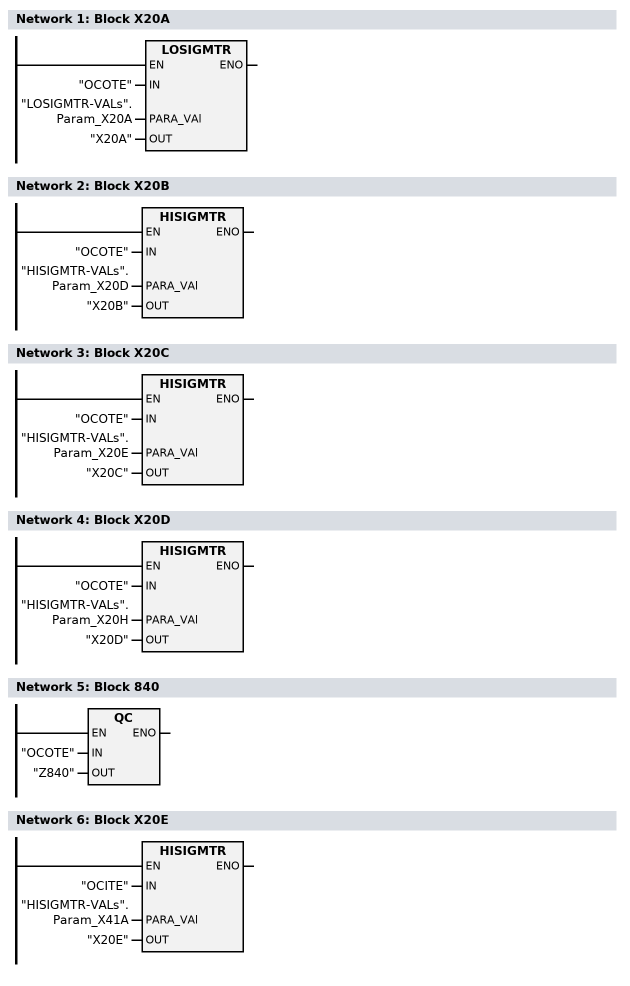
NETWORK
TITLE = Block X20A
      CALL  "LOSIGMTR" (
           IN                       := "OCOTE",
           PARA_VAl                 := "LOSIGMTR-VALs".Param_X20A,
           OUT                      := "X20A");
      NOP   0;
NETWORK
TITLE = Block X20B
      CALL  "HISIGMTR" (
           IN                       := "OCOTE",
           PARA_VAl                 := "HISIGMTR-VALs".Param_X20D,
           OUT                      := "X20B");
      NOP   0;
NETWORK
TITLE = Block X20C
      CALL  "HISIGMTR" (
           IN                       := "OCOTE",
           PARA_VAl                 := "HISIGMTR-VALs".Param_X20E,
           OUT                      := "X20C");
      NOP   0;
NETWORK
TITLE = Block X20D
      CALL  "HISIGMTR" (
           IN                       := "OCOTE",
           PARA_VAl                 := "HISIGMTR-VALs".Param_X20H,
           OUT                      := "X20D");
      NOP   0;
NETWORK
TITLE = Block 840
      CALL  "QC" (
           IN                       := "OCOTE",
           OUT                      := "Z840");
      NOP   0;
NETWORK
TITLE = Block X20E
      CALL  "HISIGMTR" (
           IN                       := "OCITE",
           PARA_VAl                 := "HISIGMTR-VALs".Param_X41A,
           OUT                      := "X20E");
      NOP   0;
END_FUNCTION

FUNCTION "2xHISIGMTV, QC" : VOID	// FC 89
TITLE = 2xHISIGMTV, QC
//Supporting block for sheet 12 (ATC)
AUTHOR : RJ
VERSION : 0.0
VAR_INPUT
  INPUT : REAL ;
  STPT_1 : REAL ;
  STPT_2 : REAL ;
  Param_1 : STRUCT
   DBAN : REAL ;
  END_STRUCT ;
  Param_2 : STRUCT
   DBAN : REAL ;
  END_STRUCT ;
END_VAR
VAR_OUTPUT
  OUT_1 : BOOL ;
  OUT_2 : BOOL ;
  OUT_QC : BOOL ;
END_VAR
VAR_TEMP
  Para_1 : STRUCT
   DBAN : REAL ;
  END_STRUCT ;
  Para_2 : STRUCT
   DBAN : REAL ;
  END_STRUCT ;
END_VAR
BEGIN
// body was compiled from an SCL source; compiled code not shown
END_FUNCTION

FUNCTION "Sheet 12 (ATC)" : VOID	// FC 91
TITLE = Sheet 12 (ATC)
//BEARING METAL TEMPERATURES (Analog)
AUTHOR : RJ
FAMILY : ATC
VERSION : 0.1
BEGIN
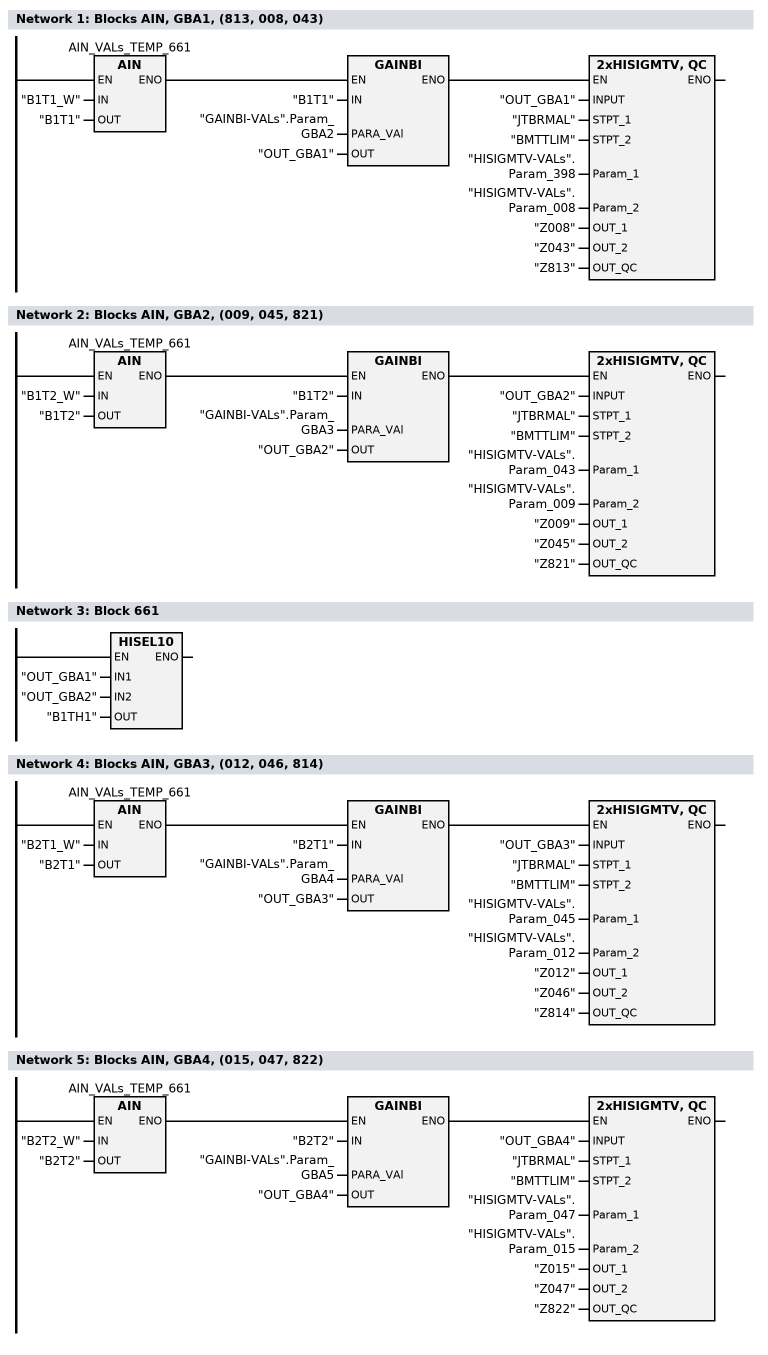
NETWORK
TITLE = Blocks AIN, GBA1, (813, 008, 043)
      A(;
      A(;
      CALL  "AIN" , "AIN_VALs_TEMP_661" (
           IN                       := "B1T1_W",
           OUT                      := "B1T1");
      A     BR;
      );
      JNB   _001;
      CALL  "GAINBI" (
           IN                       := "B1T1",
           PARA_VAl                 := "GAINBI-VALs".Param_GBA2,
           OUT                      := "OUT_GBA1");
_001: A     BR;
      );
      JNB   _002;
      CALL  "2xHISIGMTV, QC" (
           INPUT                    := "OUT_GBA1",
           STPT_1                   := "JTBRMAL",
           STPT_2                   := "BMTTLIM",
           Param_1                  := "HISIGMTV-VALs".Param_398,
           Param_2                  := "HISIGMTV-VALs".Param_008,
           OUT_1                    := "Z008",
           OUT_2                    := "Z043",
           OUT_QC                   := "Z813");
_002: NOP   0;
NETWORK
TITLE = Blocks AIN, GBA2, (009, 045, 821)
      A(;
      A(;
      CALL  "AIN" , "AIN_VALs_TEMP_661" (
           IN                       := "B1T2_W",
           OUT                      := "B1T2");
      A     BR;
      );
      JNB   _003;
      CALL  "GAINBI" (
           IN                       := "B1T2",
           PARA_VAl                 := "GAINBI-VALs".Param_GBA3,
           OUT                      := "OUT_GBA2");
_003: A     BR;
      );
      JNB   _004;
      CALL  "2xHISIGMTV, QC" (
           INPUT                    := "OUT_GBA2",
           STPT_1                   := "JTBRMAL",
           STPT_2                   := "BMTTLIM",
           Param_1                  := "HISIGMTV-VALs".Param_043,
           Param_2                  := "HISIGMTV-VALs".Param_009,
           OUT_1                    := "Z009",
           OUT_2                    := "Z045",
           OUT_QC                   := "Z821");
_004: NOP   0;
NETWORK
TITLE = Block 661
      CALL  "HISEL10" (
           IN1                      := "OUT_GBA1",
           IN2                      := "OUT_GBA2",
           OUT                      := "B1TH1");
      NOP   0;
NETWORK
TITLE = Blocks AIN, GBA3, (012, 046, 814)
      A(;
      A(;
      CALL  "AIN" , "AIN_VALs_TEMP_661" (
           IN                       := "B2T1_W",
           OUT                      := "B2T1");
      A     BR;
      );
      JNB   _005;
      CALL  "GAINBI" (
           IN                       := "B2T1",
           PARA_VAl                 := "GAINBI-VALs".Param_GBA4,
           OUT                      := "OUT_GBA3");
_005: A     BR;
      );
      JNB   _006;
      CALL  "2xHISIGMTV, QC" (
           INPUT                    := "OUT_GBA3",
           STPT_1                   := "JTBRMAL",
           STPT_2                   := "BMTTLIM",
           Param_1                  := "HISIGMTV-VALs".Param_045,
           Param_2                  := "HISIGMTV-VALs".Param_012,
           OUT_1                    := "Z012",
           OUT_2                    := "Z046",
           OUT_QC                   := "Z814");
_006: NOP   0;
NETWORK
TITLE = Blocks AIN, GBA4, (015, 047, 822)
      A(;
      A(;
      CALL  "AIN" , "AIN_VALs_TEMP_661" (
           IN                       := "B2T2_W",
           OUT                      := "B2T2");
      A     BR;
      );
      JNB   _007;
      CALL  "GAINBI" (
           IN                       := "B2T2",
           PARA_VAl                 := "GAINBI-VALs".Param_GBA5,
           OUT                      := "OUT_GBA4");
_007: A     BR;
      );
      JNB   _008;
      CALL  "2xHISIGMTV, QC" (
           INPUT                    := "OUT_GBA4",
           STPT_1                   := "JTBRMAL",
           STPT_2                   := "BMTTLIM",
           Param_1                  := "HISIGMTV-VALs".Param_047,
           Param_2                  := "HISIGMTV-VALs".Param_015,
           OUT_1                    := "Z015",
           OUT_2                    := "Z047",
           OUT_QC                   := "Z822");
_008: NOP   0;
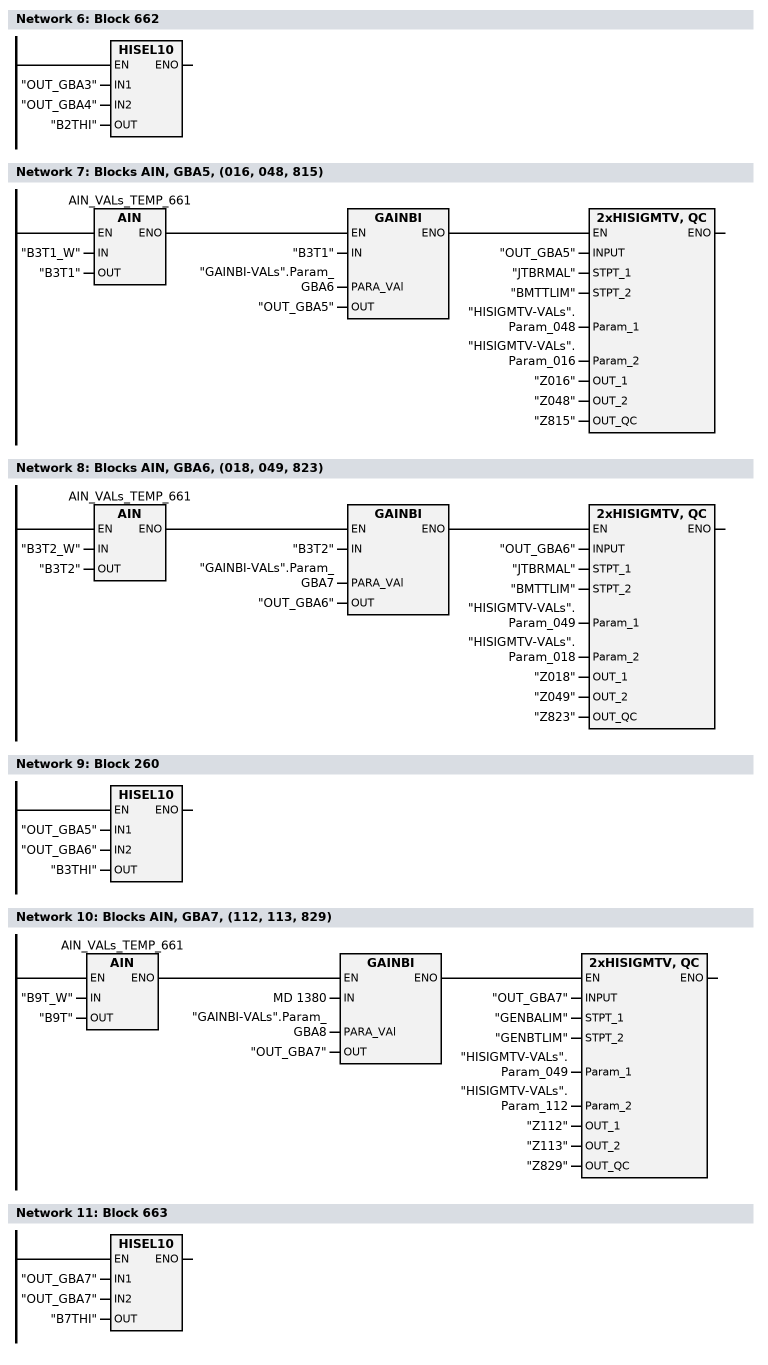
NETWORK
TITLE = Block 662
      CALL  "HISEL10" (
           IN1                      := "OUT_GBA3",
           IN2                      := "OUT_GBA4",
           OUT                      := "B2THI");
      NOP   0;
NETWORK
TITLE = Blocks AIN, GBA5, (016, 048, 815)
      A(;
      A(;
      CALL  "AIN" , "AIN_VALs_TEMP_661" (
           IN                       := "B3T1_W",
           OUT                      := "B3T1");
      A     BR;
      );
      JNB   _009;
      CALL  "GAINBI" (
           IN                       := "B3T1",
           PARA_VAl                 := "GAINBI-VALs".Param_GBA6,
           OUT                      := "OUT_GBA5");
_009: A     BR;
      );
      JNB   _00a;
      CALL  "2xHISIGMTV, QC" (
           INPUT                    := "OUT_GBA5",
           STPT_1                   := "JTBRMAL",
           STPT_2                   := "BMTTLIM",
           Param_1                  := "HISIGMTV-VALs".Param_048,
           Param_2                  := "HISIGMTV-VALs".Param_016,
           OUT_1                    := "Z016",
           OUT_2                    := "Z048",
           OUT_QC                   := "Z815");
_00a: NOP   0;
NETWORK
TITLE = Blocks AIN, GBA6, (018, 049, 823)
      A(;
      A(;
      CALL  "AIN" , "AIN_VALs_TEMP_661" (
           IN                       := "B3T2_W",
           OUT                      := "B3T2");
      A     BR;
      );
      JNB   _00b;
      CALL  "GAINBI" (
           IN                       := "B3T2",
           PARA_VAl                 := "GAINBI-VALs".Param_GBA7,
           OUT                      := "OUT_GBA6");
_00b: A     BR;
      );
      JNB   _00c;
      CALL  "2xHISIGMTV, QC" (
           INPUT                    := "OUT_GBA6",
           STPT_1                   := "JTBRMAL",
           STPT_2                   := "BMTTLIM",
           Param_1                  := "HISIGMTV-VALs".Param_049,
           Param_2                  := "HISIGMTV-VALs".Param_018,
           OUT_1                    := "Z018",
           OUT_2                    := "Z049",
           OUT_QC                   := "Z823");
_00c: NOP   0;
NETWORK
TITLE = Block 260
      CALL  "HISEL10" (
           IN1                      := "OUT_GBA5",
           IN2                      := "OUT_GBA6",
           OUT                      := "B3THI");
      NOP   0;
NETWORK
TITLE = Blocks AIN, GBA7, (112, 113, 829)
      A(;
      A(;
      CALL  "AIN" , "AIN_VALs_TEMP_661" (
           IN                       := "B9T_W",
           OUT                      := "B9T");
      A     BR;
      );
      JNB   _00d;
      CALL  "GAINBI" (
           IN                       := MD 1380,
           PARA_VAl                 := "GAINBI-VALs".Param_GBA8,
           OUT                      := "OUT_GBA7");
_00d: A     BR;
      );
      JNB   _00e;
      CALL  "2xHISIGMTV, QC" (
           INPUT                    := "OUT_GBA7",
           STPT_1                   := "GENBALIM",
           STPT_2                   := "GENBTLIM",
           Param_1                  := "HISIGMTV-VALs".Param_049,
           Param_2                  := "HISIGMTV-VALs".Param_112,
           OUT_1                    := "Z112",
           OUT_2                    := "Z113",
           OUT_QC                   := "Z829");
_00e: NOP   0;
NETWORK
TITLE = Block 663
      CALL  "HISEL10" (
           IN1                      := "OUT_GBA7",
           IN2                      := "OUT_GBA7",
           OUT                      := "B7THI");
      NOP   0;
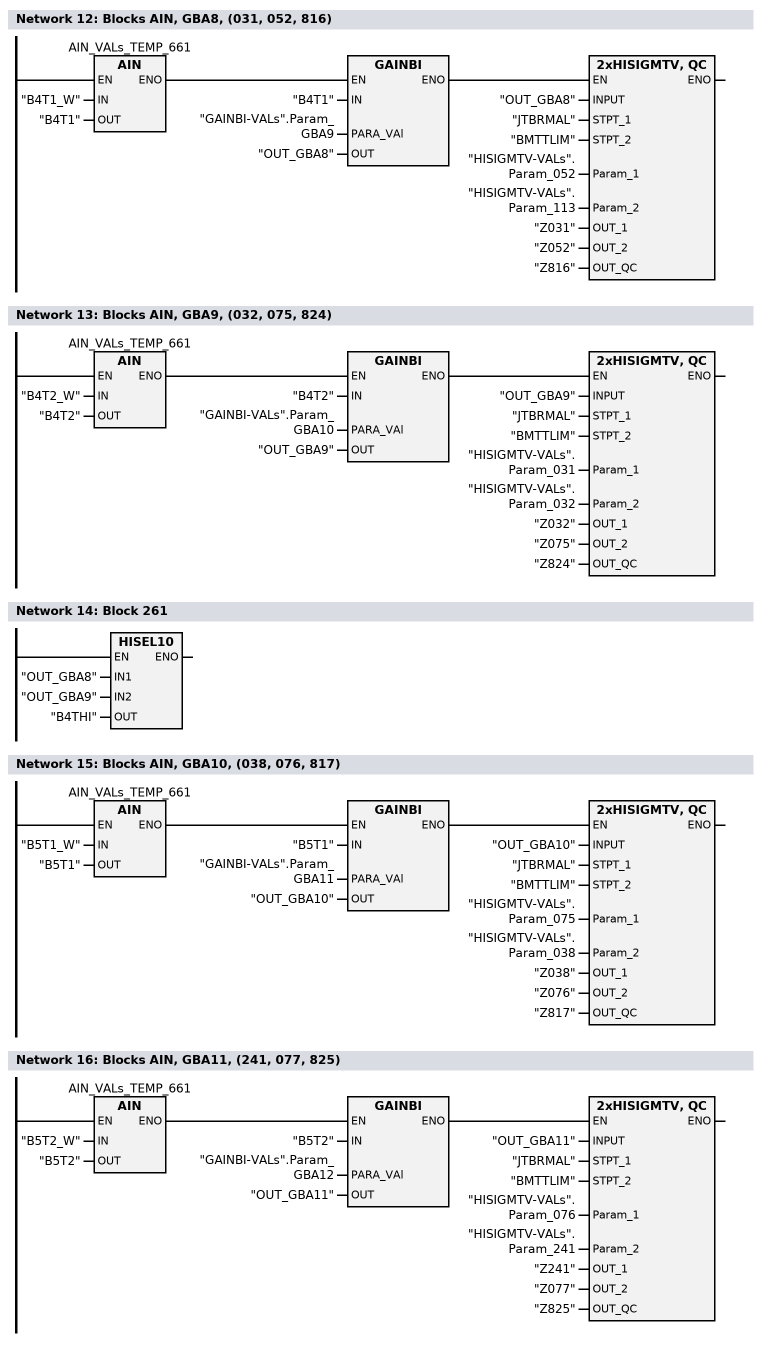
NETWORK
TITLE = Blocks AIN, GBA8, (031, 052, 816)
      A(;
      A(;
      CALL  "AIN" , "AIN_VALs_TEMP_661" (
           IN                       := "B4T1_W",
           OUT                      := "B4T1");
      A     BR;
      );
      JNB   _00f;
      CALL  "GAINBI" (
           IN                       := "B4T1",
           PARA_VAl                 := "GAINBI-VALs".Param_GBA9,
           OUT                      := "OUT_GBA8");
_00f: A     BR;
      );
      JNB   _010;
      CALL  "2xHISIGMTV, QC" (
           INPUT                    := "OUT_GBA8",
           STPT_1                   := "JTBRMAL",
           STPT_2                   := "BMTTLIM",
           Param_1                  := "HISIGMTV-VALs".Param_052,
           Param_2                  := "HISIGMTV-VALs".Param_113,
           OUT_1                    := "Z031",
           OUT_2                    := "Z052",
           OUT_QC                   := "Z816");
_010: NOP   0;
NETWORK
TITLE = Blocks AIN, GBA9, (032, 075, 824)
      A(;
      A(;
      CALL  "AIN" , "AIN_VALs_TEMP_661" (
           IN                       := "B4T2_W",
           OUT                      := "B4T2");
      A     BR;
      );
      JNB   _011;
      CALL  "GAINBI" (
           IN                       := "B4T2",
           PARA_VAl                 := "GAINBI-VALs".Param_GBA10,
           OUT                      := "OUT_GBA9");
_011: A     BR;
      );
      JNB   _012;
      CALL  "2xHISIGMTV, QC" (
           INPUT                    := "OUT_GBA9",
           STPT_1                   := "JTBRMAL",
           STPT_2                   := "BMTTLIM",
           Param_1                  := "HISIGMTV-VALs".Param_031,
           Param_2                  := "HISIGMTV-VALs".Param_032,
           OUT_1                    := "Z032",
           OUT_2                    := "Z075",
           OUT_QC                   := "Z824");
_012: NOP   0;
NETWORK
TITLE = Block 261
      CALL  "HISEL10" (
           IN1                      := "OUT_GBA8",
           IN2                      := "OUT_GBA9",
           OUT                      := "B4THI");
      NOP   0;
NETWORK
TITLE = Blocks AIN, GBA10, (038, 076, 817)
      A(;
      A(;
      CALL  "AIN" , "AIN_VALs_TEMP_661" (
           IN                       := "B5T1_W",
           OUT                      := "B5T1");
      A     BR;
      );
      JNB   _013;
      CALL  "GAINBI" (
           IN                       := "B5T1",
           PARA_VAl                 := "GAINBI-VALs".Param_GBA11,
           OUT                      := "OUT_GBA10");
_013: A     BR;
      );
      JNB   _014;
      CALL  "2xHISIGMTV, QC" (
           INPUT                    := "OUT_GBA10",
           STPT_1                   := "JTBRMAL",
           STPT_2                   := "BMTTLIM",
           Param_1                  := "HISIGMTV-VALs".Param_075,
           Param_2                  := "HISIGMTV-VALs".Param_038,
           OUT_1                    := "Z038",
           OUT_2                    := "Z076",
           OUT_QC                   := "Z817");
_014: NOP   0;
NETWORK
TITLE = Blocks AIN, GBA11, (241, 077, 825)
      A(;
      A(;
      CALL  "AIN" , "AIN_VALs_TEMP_661" (
           IN                       := "B5T2_W",
           OUT                      := "B5T2");
      A     BR;
      );
      JNB   _015;
      CALL  "GAINBI" (
           IN                       := "B5T2",
           PARA_VAl                 := "GAINBI-VALs".Param_GBA12,
           OUT                      := "OUT_GBA11");
_015: A     BR;
      );
      JNB   _016;
      CALL  "2xHISIGMTV, QC" (
           INPUT                    := "OUT_GBA11",
           STPT_1                   := "JTBRMAL",
           STPT_2                   := "BMTTLIM",
           Param_1                  := "HISIGMTV-VALs".Param_076,
           Param_2                  := "HISIGMTV-VALs".Param_241,
           OUT_1                    := "Z241",
           OUT_2                    := "Z077",
           OUT_QC                   := "Z825");
_016: NOP   0;
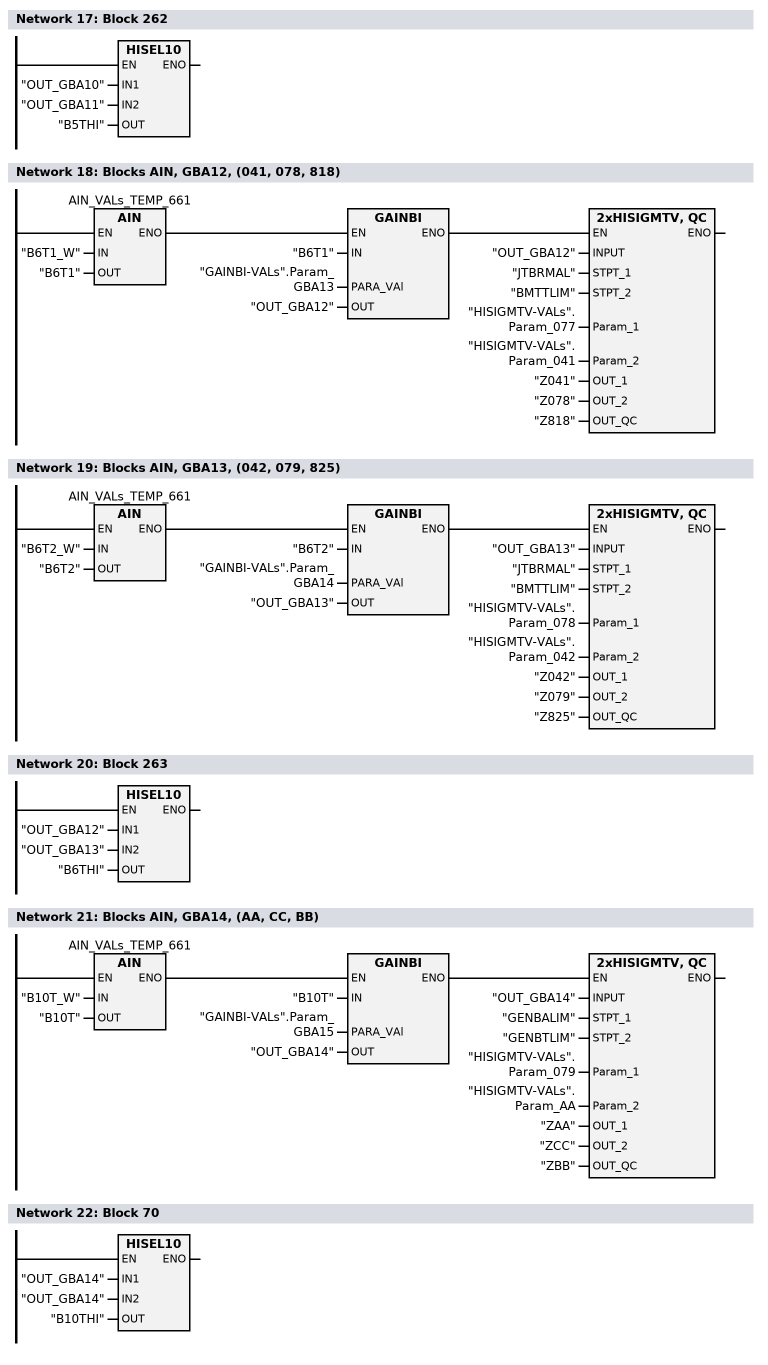
NETWORK
TITLE = Block 262
      CALL  "HISEL10" (
           IN1                      := "OUT_GBA10",
           IN2                      := "OUT_GBA11",
           OUT                      := "B5THI");
      NOP   0;
NETWORK
TITLE = Blocks AIN, GBA12, (041, 078, 818)
      A(;
      A(;
      CALL  "AIN" , "AIN_VALs_TEMP_661" (
           IN                       := "B6T1_W",
           OUT                      := "B6T1");
      A     BR;
      );
      JNB   _017;
      CALL  "GAINBI" (
           IN                       := "B6T1",
           PARA_VAl                 := "GAINBI-VALs".Param_GBA13,
           OUT                      := "OUT_GBA12");
_017: A     BR;
      );
      JNB   _018;
      CALL  "2xHISIGMTV, QC" (
           INPUT                    := "OUT_GBA12",
           STPT_1                   := "JTBRMAL",
           STPT_2                   := "BMTTLIM",
           Param_1                  := "HISIGMTV-VALs".Param_077,
           Param_2                  := "HISIGMTV-VALs".Param_041,
           OUT_1                    := "Z041",
           OUT_2                    := "Z078",
           OUT_QC                   := "Z818");
_018: NOP   0;
NETWORK
TITLE = Blocks AIN, GBA13, (042, 079, 825)
      A(;
      A(;
      CALL  "AIN" , "AIN_VALs_TEMP_661" (
           IN                       := "B6T2_W",
           OUT                      := "B6T2");
      A     BR;
      );
      JNB   _019;
      CALL  "GAINBI" (
           IN                       := "B6T2",
           PARA_VAl                 := "GAINBI-VALs".Param_GBA14,
           OUT                      := "OUT_GBA13");
_019: A     BR;
      );
      JNB   _01a;
      CALL  "2xHISIGMTV, QC" (
           INPUT                    := "OUT_GBA13",
           STPT_1                   := "JTBRMAL",
           STPT_2                   := "BMTTLIM",
           Param_1                  := "HISIGMTV-VALs".Param_078,
           Param_2                  := "HISIGMTV-VALs".Param_042,
           OUT_1                    := "Z042",
           OUT_2                    := "Z079",
           OUT_QC                   := "Z825");
_01a: NOP   0;
NETWORK
TITLE = Block 263
      CALL  "HISEL10" (
           IN1                      := "OUT_GBA12",
           IN2                      := "OUT_GBA13",
           OUT                      := "B6THI");
      NOP   0;
NETWORK
TITLE = Blocks AIN, GBA14, (AA, CC, BB)
      A(;
      A(;
      CALL  "AIN" , "AIN_VALs_TEMP_661" (
           IN                       := "B10T_W",
           OUT                      := "B10T");
      A     BR;
      );
      JNB   _01b;
      CALL  "GAINBI" (
           IN                       := "B10T",
           PARA_VAl                 := "GAINBI-VALs".Param_GBA15,
           OUT                      := "OUT_GBA14");
_01b: A     BR;
      );
      JNB   _01c;
      CALL  "2xHISIGMTV, QC" (
           INPUT                    := "OUT_GBA14",
           STPT_1                   := "GENBALIM",
           STPT_2                   := "GENBTLIM",
           Param_1                  := "HISIGMTV-VALs".Param_079,
           Param_2                  := "HISIGMTV-VALs".Param_AA,
           OUT_1                    := "ZAA",
           OUT_2                    := "ZCC",
           OUT_QC                   := "ZBB");
_01c: NOP   0;
NETWORK
TITLE = Block 70
      CALL  "HISEL10" (
           IN1                      := "OUT_GBA14",
           IN2                      := "OUT_GBA14",
           OUT                      := "B10THI");
      NOP   0;
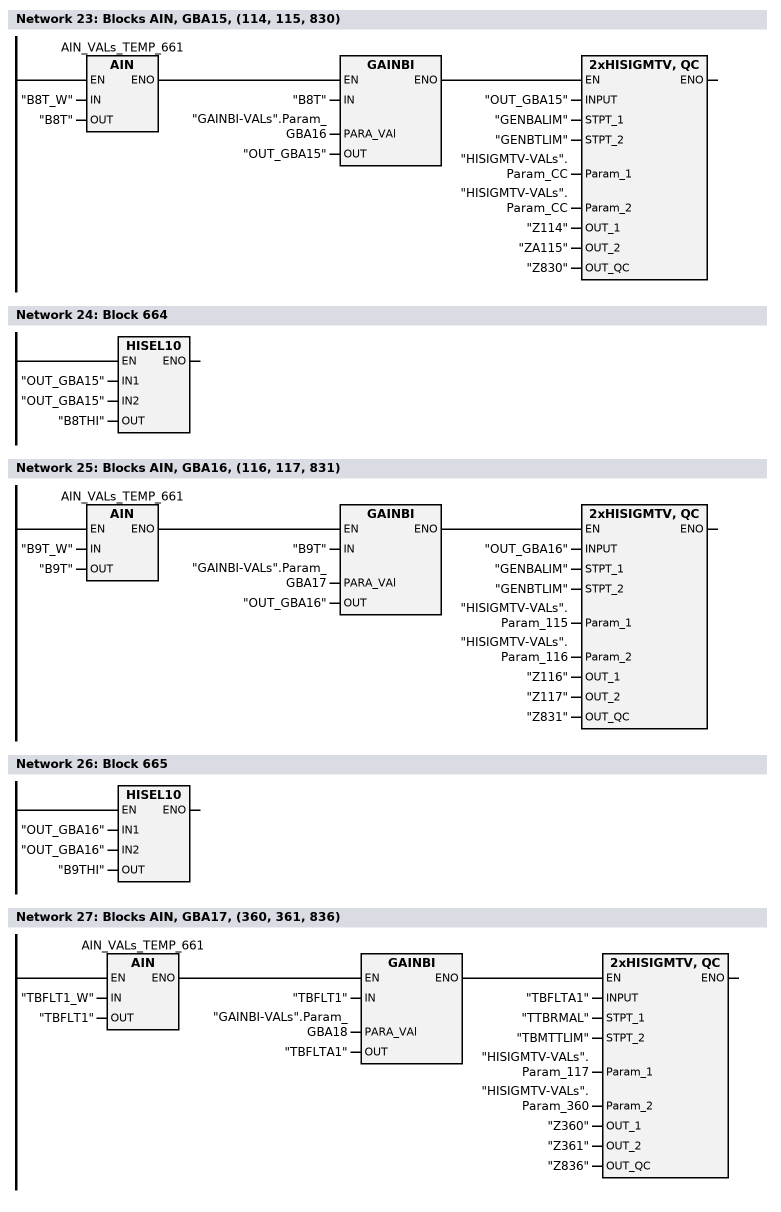
NETWORK
TITLE = Blocks AIN, GBA15, (114, 115, 830)
      A(;
      A(;
      CALL  "AIN" , "AIN_VALs_TEMP_661" (
           IN                       := "B8T_W",
           OUT                      := "B8T");
      A     BR;
      );
      JNB   _01d;
      CALL  "GAINBI" (
           IN                       := "B8T",
           PARA_VAl                 := "GAINBI-VALs".Param_GBA16,
           OUT                      := "OUT_GBA15");
_01d: A     BR;
      );
      JNB   _01e;
      CALL  "2xHISIGMTV, QC" (
           INPUT                    := "OUT_GBA15",
           STPT_1                   := "GENBALIM",
           STPT_2                   := "GENBTLIM",
           Param_1                  := "HISIGMTV-VALs".Param_CC,
           Param_2                  := "HISIGMTV-VALs".Param_CC,
           OUT_1                    := "Z114",
           OUT_2                    := "ZA115",
           OUT_QC                   := "Z830");
_01e: NOP   0;
NETWORK
TITLE = Block 664
      CALL  "HISEL10" (
           IN1                      := "OUT_GBA15",
           IN2                      := "OUT_GBA15",
           OUT                      := "B8THI");
      NOP   0;
NETWORK
TITLE = Blocks AIN, GBA16, (116, 117, 831)
      A(;
      A(;
      CALL  "AIN" , "AIN_VALs_TEMP_661" (
           IN                       := "B9T_W",
           OUT                      := "B9T");
      A     BR;
      );
      JNB   _01f;
      CALL  "GAINBI" (
           IN                       := "B9T",
           PARA_VAl                 := "GAINBI-VALs".Param_GBA17,
           OUT                      := "OUT_GBA16");
_01f: A     BR;
      );
      JNB   _020;
      CALL  "2xHISIGMTV, QC" (
           INPUT                    := "OUT_GBA16",
           STPT_1                   := "GENBALIM",
           STPT_2                   := "GENBTLIM",
           Param_1                  := "HISIGMTV-VALs".Param_115,
           Param_2                  := "HISIGMTV-VALs".Param_116,
           OUT_1                    := "Z116",
           OUT_2                    := "Z117",
           OUT_QC                   := "Z831");
_020: NOP   0;
NETWORK
TITLE = Block 665
      CALL  "HISEL10" (
           IN1                      := "OUT_GBA16",
           IN2                      := "OUT_GBA16",
           OUT                      := "B9THI");
      NOP   0;
NETWORK
TITLE = Blocks AIN, GBA17, (360, 361, 836)
      A(;
      A(;
      CALL  "AIN" , "AIN_VALs_TEMP_661" (
           IN                       := "TBFLT1_W",
           OUT                      := "TBFLT1");
      A     BR;
      );
      JNB   _021;
      CALL  "GAINBI" (
           IN                       := "TBFLT1",
           PARA_VAl                 := "GAINBI-VALs".Param_GBA18,
           OUT                      := "TBFLTA1");
_021: A     BR;
      );
      JNB   _022;
      CALL  "2xHISIGMTV, QC" (
           INPUT                    := "TBFLTA1",
           STPT_1                   := "TTBRMAL",
           STPT_2                   := "TBMTTLIM",
           Param_1                  := "HISIGMTV-VALs".Param_117,
           Param_2                  := "HISIGMTV-VALs".Param_360,
           OUT_1                    := "Z360",
           OUT_2                    := "Z361",
           OUT_QC                   := "Z836");
_022: NOP   0;
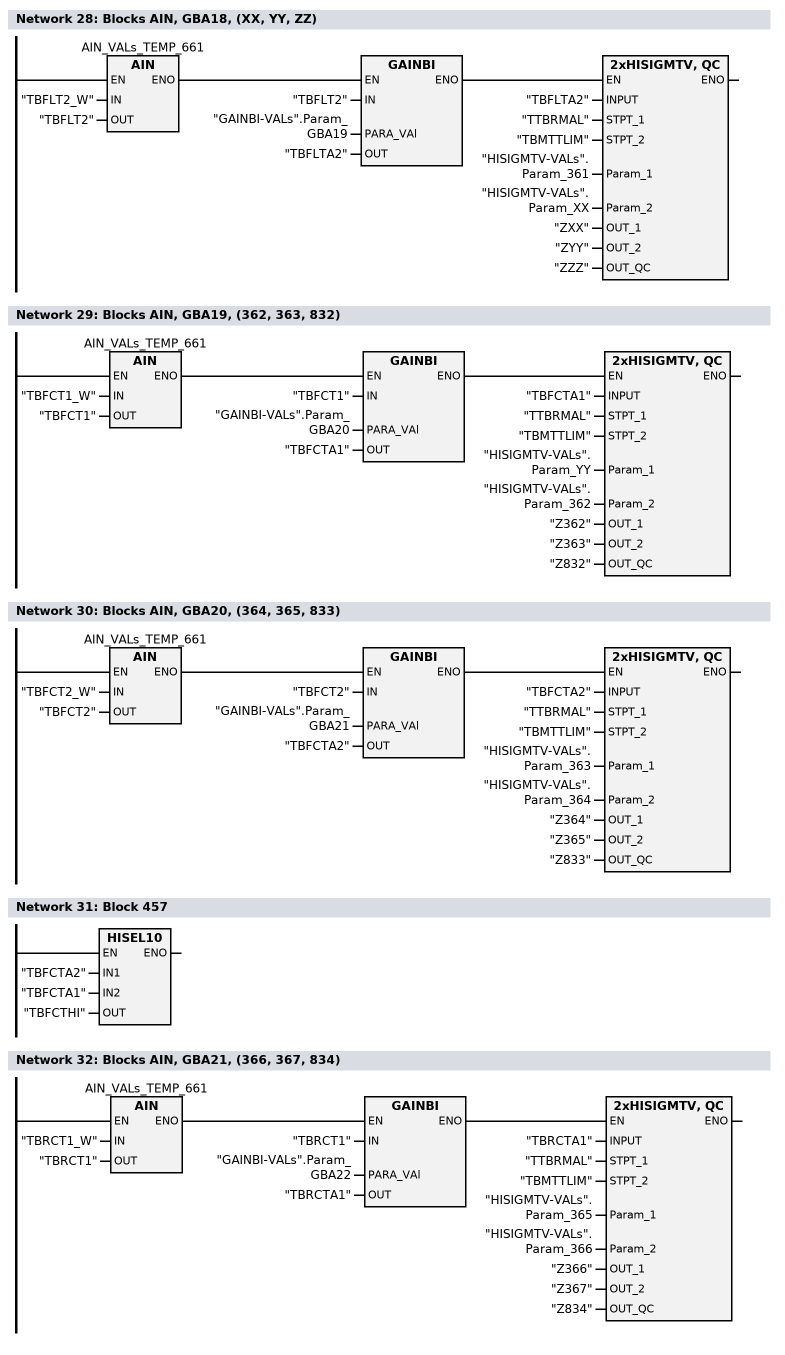
NETWORK
TITLE = Blocks AIN, GBA18, (XX, YY, ZZ)
      A(;
      A(;
      CALL  "AIN" , "AIN_VALs_TEMP_661" (
           IN                       := "TBFLT2_W",
           OUT                      := "TBFLT2");
      A     BR;
      );
      JNB   _023;
      CALL  "GAINBI" (
           IN                       := "TBFLT2",
           PARA_VAl                 := "GAINBI-VALs".Param_GBA19,
           OUT                      := "TBFLTA2");
_023: A     BR;
      );
      JNB   _024;
      CALL  "2xHISIGMTV, QC" (
           INPUT                    := "TBFLTA2",
           STPT_1                   := "TTBRMAL",
           STPT_2                   := "TBMTTLIM",
           Param_1                  := "HISIGMTV-VALs".Param_361,
           Param_2                  := "HISIGMTV-VALs".Param_XX,
           OUT_1                    := "ZXX",
           OUT_2                    := "ZYY",
           OUT_QC                   := "ZZZ");
_024: NOP   0;
NETWORK
TITLE = Blocks AIN, GBA19, (362, 363, 832)
      A(;
      A(;
      CALL  "AIN" , "AIN_VALs_TEMP_661" (
           IN                       := "TBFCT1_W",
           OUT                      := "TBFCT1");
      A     BR;
      );
      JNB   _025;
      CALL  "GAINBI" (
           IN                       := "TBFCT1",
           PARA_VAl                 := "GAINBI-VALs".Param_GBA20,
           OUT                      := "TBFCTA1");
_025: A     BR;
      );
      JNB   _026;
      CALL  "2xHISIGMTV, QC" (
           INPUT                    := "TBFCTA1",
           STPT_1                   := "TTBRMAL",
           STPT_2                   := "TBMTTLIM",
           Param_1                  := "HISIGMTV-VALs".Param_YY,
           Param_2                  := "HISIGMTV-VALs".Param_362,
           OUT_1                    := "Z362",
           OUT_2                    := "Z363",
           OUT_QC                   := "Z832");
_026: NOP   0;
NETWORK
TITLE = Blocks AIN, GBA20, (364, 365, 833)
      A(;
      A(;
      CALL  "AIN" , "AIN_VALs_TEMP_661" (
           IN                       := "TBFCT2_W",
           OUT                      := "TBFCT2");
      A     BR;
      );
      JNB   _027;
      CALL  "GAINBI" (
           IN                       := "TBFCT2",
           PARA_VAl                 := "GAINBI-VALs".Param_GBA21,
           OUT                      := "TBFCTA2");
_027: A     BR;
      );
      JNB   _028;
      CALL  "2xHISIGMTV, QC" (
           INPUT                    := "TBFCTA2",
           STPT_1                   := "TTBRMAL",
           STPT_2                   := "TBMTTLIM",
           Param_1                  := "HISIGMTV-VALs".Param_363,
           Param_2                  := "HISIGMTV-VALs".Param_364,
           OUT_1                    := "Z364",
           OUT_2                    := "Z365",
           OUT_QC                   := "Z833");
_028: NOP   0;
NETWORK
TITLE = Block 457
      CALL  "HISEL10" (
           IN1                      := "TBFCTA2",
           IN2                      := "TBFCTA1",
           OUT                      := "TBFCTHI");
      NOP   0;
NETWORK
TITLE = Blocks AIN, GBA21, (366, 367, 834)
      A(;
      A(;
      CALL  "AIN" , "AIN_VALs_TEMP_661" (
           IN                       := "TBRCT1_W",
           OUT                      := "TBRCT1");
      A     BR;
      );
      JNB   _029;
      CALL  "GAINBI" (
           IN                       := "TBRCT1",
           PARA_VAl                 := "GAINBI-VALs".Param_GBA22,
           OUT                      := "TBRCTA1");
_029: A     BR;
      );
      JNB   _02a;
      CALL  "2xHISIGMTV, QC" (
           INPUT                    := "TBRCTA1",
           STPT_1                   := "TTBRMAL",
           STPT_2                   := "TBMTTLIM",
           Param_1                  := "HISIGMTV-VALs".Param_365,
           Param_2                  := "HISIGMTV-VALs".Param_366,
           OUT_1                    := "Z366",
           OUT_2                    := "Z367",
           OUT_QC                   := "Z834");
_02a: NOP   0;
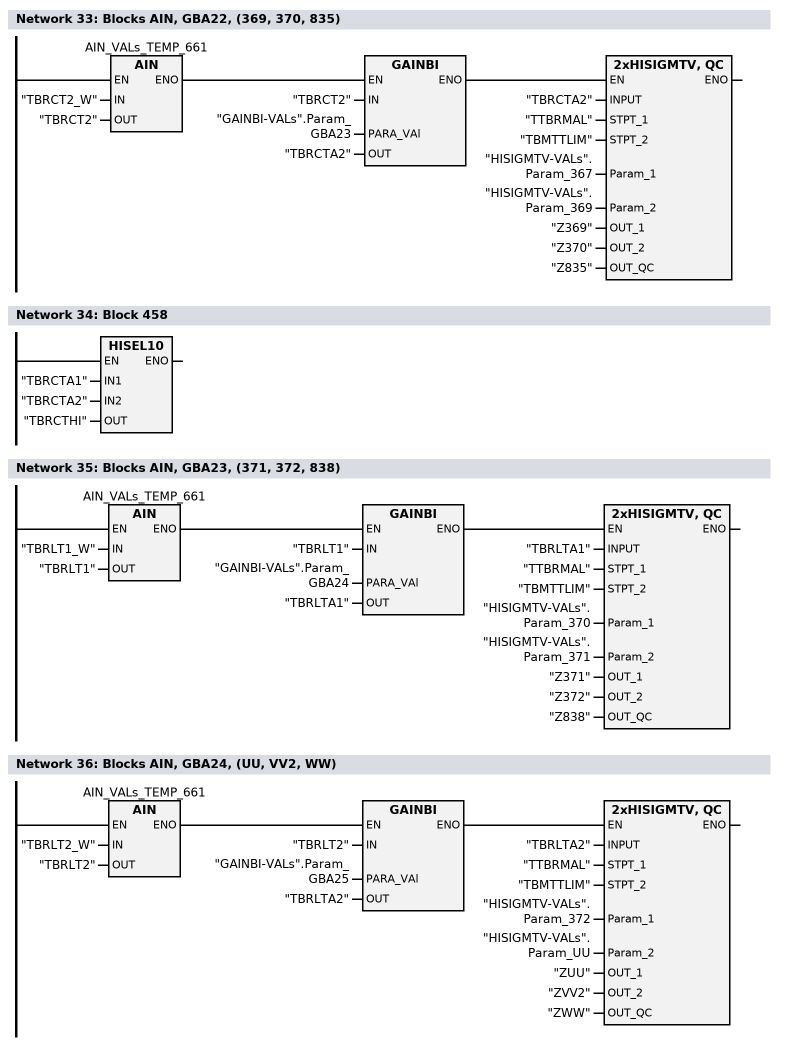
NETWORK
TITLE = Blocks AIN, GBA22, (369, 370, 835)
      A(;
      A(;
      CALL  "AIN" , "AIN_VALs_TEMP_661" (
           IN                       := "TBRCT2_W",
           OUT                      := "TBRCT2");
      A     BR;
      );
      JNB   _02b;
      CALL  "GAINBI" (
           IN                       := "TBRCT2",
           PARA_VAl                 := "GAINBI-VALs".Param_GBA23,
           OUT                      := "TBRCTA2");
_02b: A     BR;
      );
      JNB   _02c;
      CALL  "2xHISIGMTV, QC" (
           INPUT                    := "TBRCTA2",
           STPT_1                   := "TTBRMAL",
           STPT_2                   := "TBMTTLIM",
           Param_1                  := "HISIGMTV-VALs".Param_367,
           Param_2                  := "HISIGMTV-VALs".Param_369,
           OUT_1                    := "Z369",
           OUT_2                    := "Z370",
           OUT_QC                   := "Z835");
_02c: NOP   0;
NETWORK
TITLE = Block 458
      CALL  "HISEL10" (
           IN1                      := "TBRCTA1",
           IN2                      := "TBRCTA2",
           OUT                      := "TBRCTHI");
      NOP   0;
NETWORK
TITLE = Blocks AIN, GBA23, (371, 372, 838)
      A(;
      A(;
      CALL  "AIN" , "AIN_VALs_TEMP_661" (
           IN                       := "TBRLT1_W",
           OUT                      := "TBRLT1");
      A     BR;
      );
      JNB   _02d;
      CALL  "GAINBI" (
           IN                       := "TBRLT1",
           PARA_VAl                 := "GAINBI-VALs".Param_GBA24,
           OUT                      := "TBRLTA1");
_02d: A     BR;
      );
      JNB   _02e;
      CALL  "2xHISIGMTV, QC" (
           INPUT                    := "TBRLTA1",
           STPT_1                   := "TTBRMAL",
           STPT_2                   := "TBMTTLIM",
           Param_1                  := "HISIGMTV-VALs".Param_370,
           Param_2                  := "HISIGMTV-VALs".Param_371,
           OUT_1                    := "Z371",
           OUT_2                    := "Z372",
           OUT_QC                   := "Z838");
_02e: NOP   0;
NETWORK
TITLE = Blocks AIN, GBA24, (UU, VV2, WW)
      A(;
      A(;
      CALL  "AIN" , "AIN_VALs_TEMP_661" (
           IN                       := "TBRLT2_W",
           OUT                      := "TBRLT2");
      A     BR;
      );
      JNB   _02f;
      CALL  "GAINBI" (
           IN                       := "TBRLT2",
           PARA_VAl                 := "GAINBI-VALs".Param_GBA25,
           OUT                      := "TBRLTA2");
_02f: A     BR;
      );
      JNB   _030;
      CALL  "2xHISIGMTV, QC" (
           INPUT                    := "TBRLTA2",
           STPT_1                   := "TTBRMAL",
           STPT_2                   := "TBMTTLIM",
           Param_1                  := "HISIGMTV-VALs".Param_372,
           Param_2                  := "HISIGMTV-VALs".Param_UU,
           OUT_1                    := "ZUU",
           OUT_2                    := "ZVV2",
           OUT_QC                   := "ZWW");
_030: NOP   0;
END_FUNCTION

FUNCTION "Sheet 13 (ATC)" : VOID	// FC 92
TITLE = Sheet 13 (ATC)
//BEARING METAL, OIL COOLER - P08MXX (Digital)
AUTHOR : RJ
FAMILY : ATC
VERSION : 0.1
BEGIN
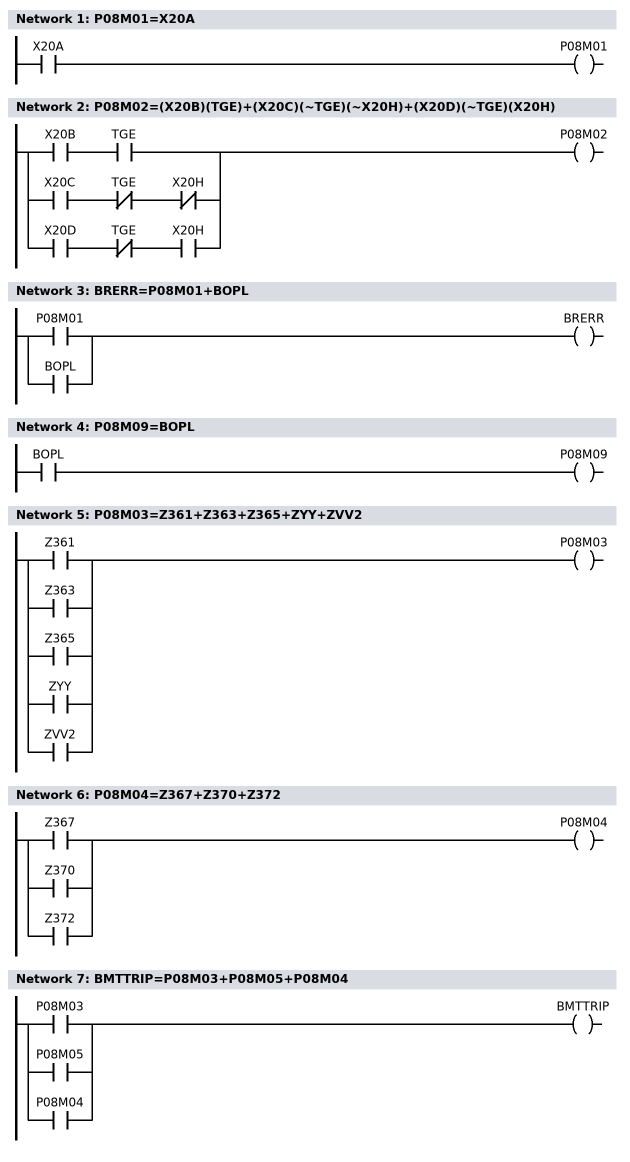
NETWORK
TITLE = P08M01=X20A
      A     "X20A";
      =     "P08M01";
NETWORK
TITLE = P08M02=(X20B)(TGE)+(X20C)(~TGE)(~X20H)+(X20D)(~TGE)(X20H)
      A     "X20B";
      A     "TGE";
      O;
      A     "X20C";
      AN    "TGE";
      AN    "X20H";
      O;
      A     "X20D";
      AN    "TGE";
      A     "X20H";
      =     "P08M02";
NETWORK
TITLE = BRERR=P08M01+BOPL
      O     "P08M01";
      O     "BOPL";
      =     "BRERR";
NETWORK
TITLE = P08M09=BOPL
      A     "BOPL";
      =     "P08M09";
NETWORK
TITLE = P08M03=Z361+Z363+Z365+ZYY+ZVV2
      O     "Z361";
      O     "Z363";
      O     "Z365";
      O     "ZYY";
      O     "ZVV2";
      =     "P08M03";
NETWORK
TITLE = P08M04=Z367+Z370+Z372
      O     "Z367";
      O     "Z370";
      O     "Z372";
      =     "P08M04";
NETWORK
TITLE = BMTTRIP=P08M03+P08M05+P08M04
      O     "P08M03";
      O     "P08M05";
      O     "P08M04";
      =     "BMTTRIP";
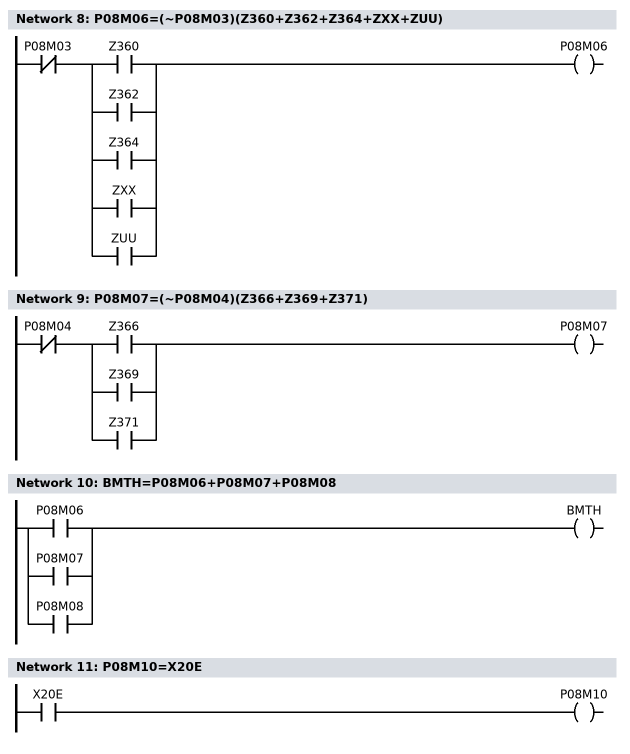
NETWORK
TITLE = P08M06=(~P08M03)(Z360+Z362+Z364+ZXX+ZUU)
      AN    "P08M03";
      A(;
      O     "Z360";
      O     "Z362";
      O     "Z364";
      O     "ZXX";
      O     "ZUU";
      );
      =     "P08M06";
NETWORK
TITLE = P08M07=(~P08M04)(Z366+Z369+Z371)
      AN    "P08M04";
      A(;
      O     "Z366";
      O     "Z369";
      O     "Z371";
      );
      =     "P08M07";
NETWORK
TITLE = BMTH=P08M06+P08M07+P08M08
      O     "P08M06";
      O     "P08M07";
      O     "P08M08";
      =     "BMTH";
NETWORK
TITLE = P08M10=X20E
      A     "X20E";
      =     "P08M10";
END_FUNCTION

FUNCTION "Sheet 14 (ATC)" : VOID	// FC 93
TITLE = Sheet 14 (ATC)
//BEARING METAL - P08M05, 8 (Digital)
AUTHOR : RJ
FAMILY : ATC
VERSION : 0.1
BEGIN
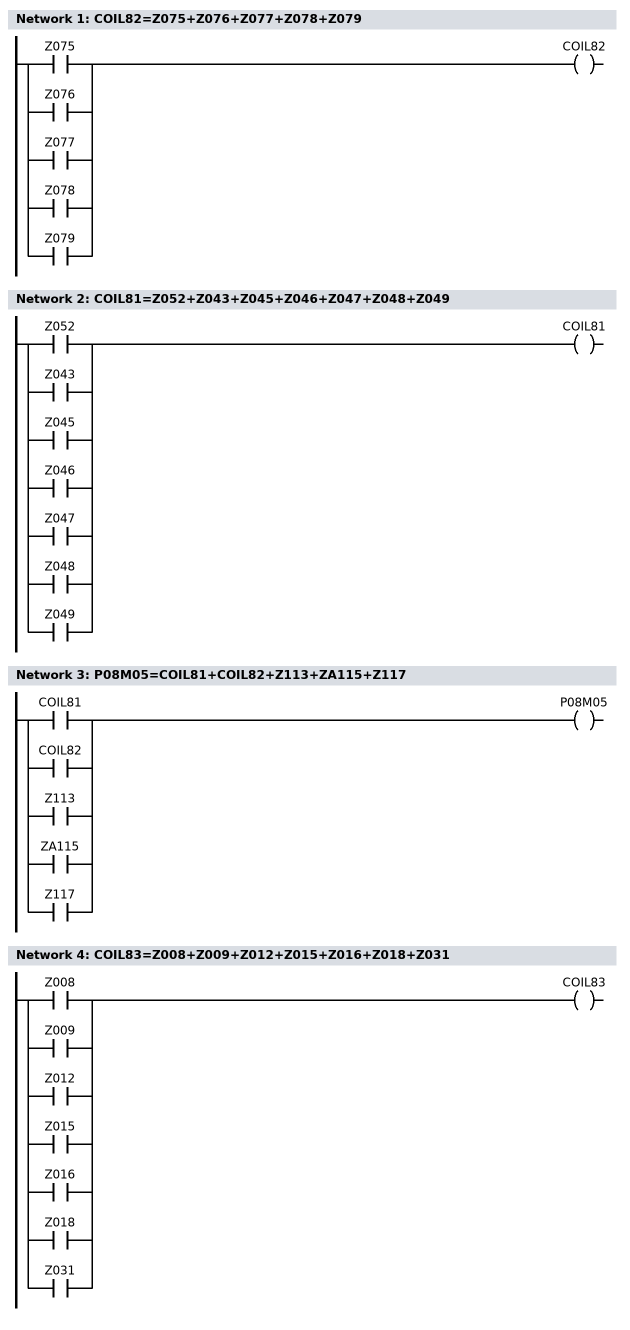
NETWORK
TITLE = COIL82=Z075+Z076+Z077+Z078+Z079
      O     "Z075";
      O     "Z076";
      O     "Z077";
      O     "Z078";
      O     "Z079";
      =     "COIL82";
NETWORK
TITLE = COIL81=Z052+Z043+Z045+Z046+Z047+Z048+Z049
      O     "Z052";
      O     "Z043";
      O     "Z045";
      O     "Z046";
      O     "Z047";
      O     "Z048";
      O     "Z049";
      =     "COIL81";
NETWORK
TITLE = P08M05=COIL81+COIL82+Z113+ZA115+Z117
      O     "COIL81";
      O     "COIL82";
      O     "Z113";
      O     "ZA115";
      O     "Z117";
      =     "P08M05";
NETWORK
TITLE = COIL83=Z008+Z009+Z012+Z015+Z016+Z018+Z031
      O     "Z008";
      O     "Z009";
      O     "Z012";
      O     "Z015";
      O     "Z016";
      O     "Z018";
      O     "Z031";
      =     "COIL83";
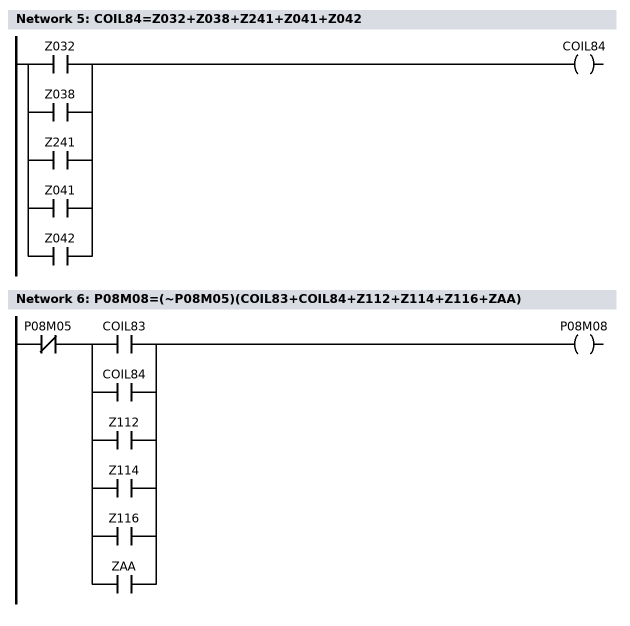
NETWORK
TITLE = COIL84=Z032+Z038+Z241+Z041+Z042
      O     "Z032";
      O     "Z038";
      O     "Z241";
      O     "Z041";
      O     "Z042";
      =     "COIL84";
NETWORK
TITLE = P08M08=(~P08M05)(COIL83+COIL84+Z112+Z114+Z116+ZAA)
      AN    "P08M05";
      A(;
      O     "COIL83";
      O     "COIL84";
      O     "Z112";
      O     "Z114";
      O     "Z116";
      O     "ZAA";
      );
      =     "P08M08";
END_FUNCTION

FUNCTION "Sheet 15 (ATC)" : VOID	// FC 94
TITLE = Sheet 15 (ATC)
//ROTOR POSITION, DIFF EXPANSION (Analog)
AUTHOR : RJ
FAMILY : ATC
VERSION : 0.1
BEGIN
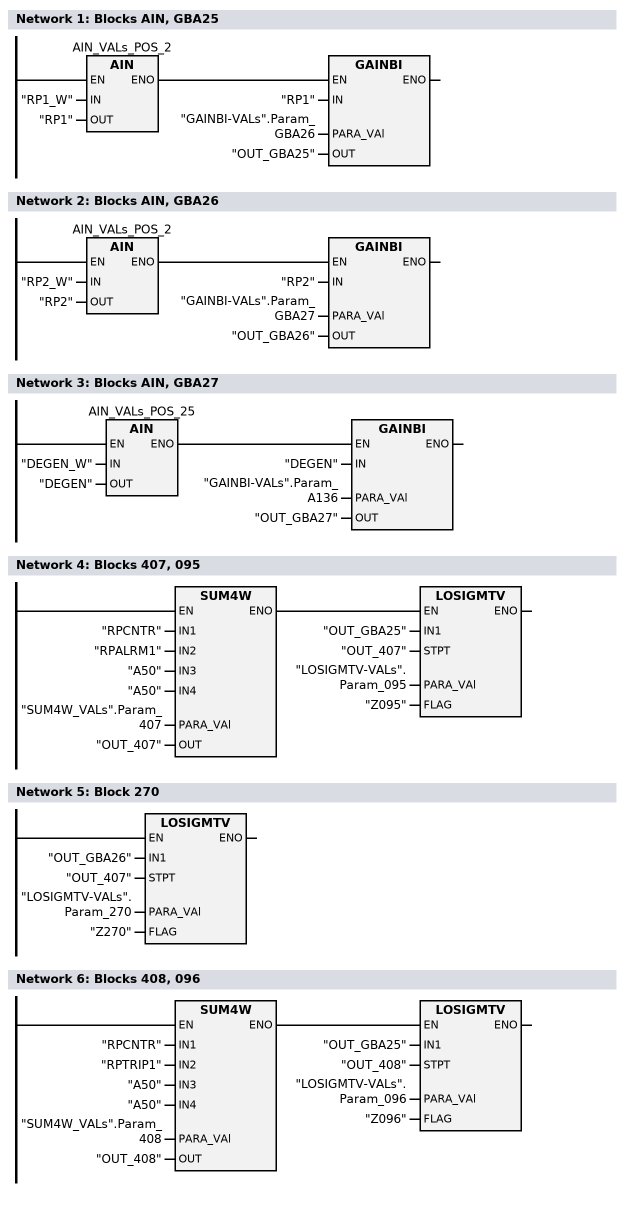
NETWORK
TITLE = Blocks AIN, GBA25
      A(;
      CALL  "AIN" , "AIN_VALs_POS_2" (
           IN                       := "RP1_W",
           OUT                      := "RP1");
      A     BR;
      );
      JNB   _001;
      CALL  "GAINBI" (
           IN                       := "RP1",
           PARA_VAl                 := "GAINBI-VALs".Param_GBA26,
           OUT                      := "OUT_GBA25");
_001: NOP   0;
NETWORK
TITLE = Blocks AIN, GBA26
      A(;
      CALL  "AIN" , "AIN_VALs_POS_2" (
           IN                       := "RP2_W",
           OUT                      := "RP2");
      A     BR;
      );
      JNB   _002;
      CALL  "GAINBI" (
           IN                       := "RP2",
           PARA_VAl                 := "GAINBI-VALs".Param_GBA27,
           OUT                      := "OUT_GBA26");
_002: NOP   0;
NETWORK
TITLE = Blocks AIN, GBA27
      A(;
      CALL  "AIN" , "AIN_VALs_POS_25" (
           IN                       := "DEGEN_W",
           OUT                      := "DEGEN");
      A     BR;
      );
      JNB   _003;
      CALL  "GAINBI" (
           IN                       := "DEGEN",
           PARA_VAl                 := "GAINBI-VALs".Param_A136,
           OUT                      := "OUT_GBA27");
_003: NOP   0;
NETWORK
TITLE = Blocks 407, 095
      A(;
      CALL  "SUM4W" (
           IN1                      := "RPCNTR",
           IN2                      := "RPALRM1",
           IN3                      := "A50",
           IN4                      := "A50",
           PARA_VAl                 := "SUM4W_VALs".Param_407,
           OUT                      := "OUT_407");
      A     BR;
      );
      JNB   _004;
      CALL  "LOSIGMTV" (
           IN1                      := "OUT_GBA25",
           STPT                     := "OUT_407",
           PARA_VAl                 := "LOSIGMTV-VALs".Param_095,
           FLAG                     := "Z095");
_004: NOP   0;
NETWORK
TITLE = Block 270
      CALL  "LOSIGMTV" (
           IN1                      := "OUT_GBA26",
           STPT                     := "OUT_407",
           PARA_VAl                 := "LOSIGMTV-VALs".Param_270,
           FLAG                     := "Z270");
      NOP   0;
NETWORK
TITLE = Blocks 408, 096
      A(;
      CALL  "SUM4W" (
           IN1                      := "RPCNTR",
           IN2                      := "RPTRIP1",
           IN3                      := "A50",
           IN4                      := "A50",
           PARA_VAl                 := "SUM4W_VALs".Param_408,
           OUT                      := "OUT_408");
      A     BR;
      );
      JNB   _005;
      CALL  "LOSIGMTV" (
           IN1                      := "OUT_GBA25",
           STPT                     := "OUT_408",
           PARA_VAl                 := "LOSIGMTV-VALs".Param_096,
           FLAG                     := "Z096");
_005: NOP   0;
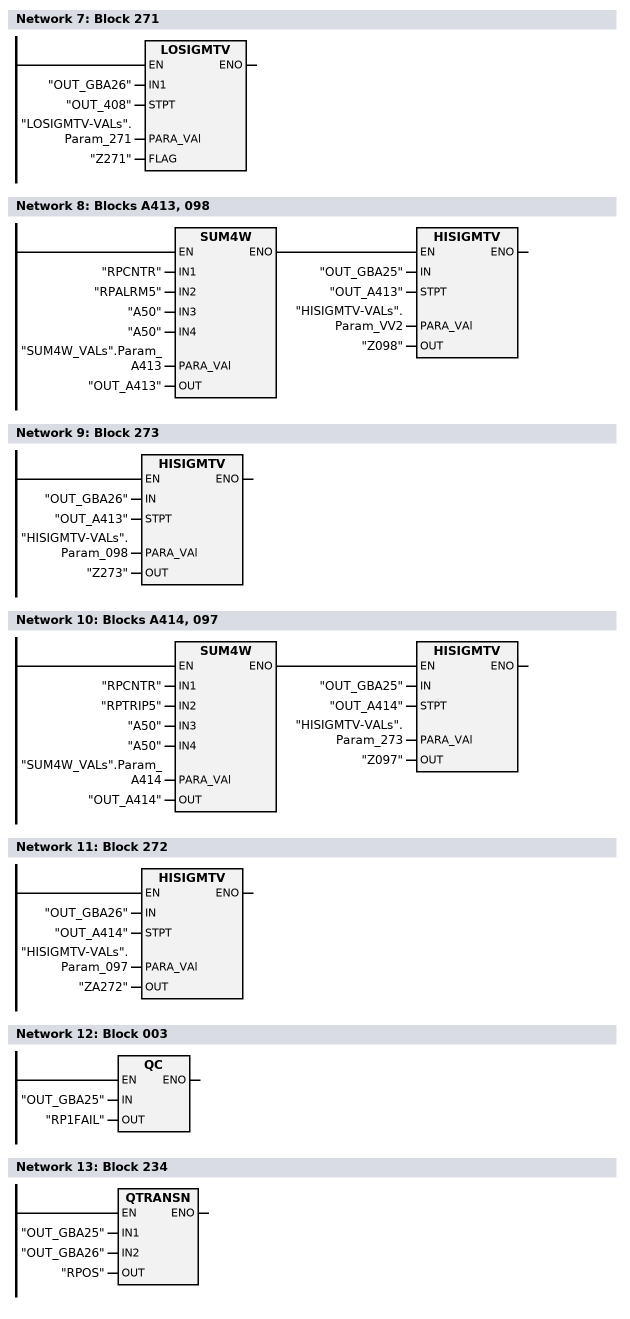
NETWORK
TITLE = Block 271
      CALL  "LOSIGMTV" (
           IN1                      := "OUT_GBA26",
           STPT                     := "OUT_408",
           PARA_VAl                 := "LOSIGMTV-VALs".Param_271,
           FLAG                     := "Z271");
      NOP   0;
NETWORK
TITLE = Blocks A413, 098
      A(;
      CALL  "SUM4W" (
           IN1                      := "RPCNTR",
           IN2                      := "RPALRM5",
           IN3                      := "A50",
           IN4                      := "A50",
           PARA_VAl                 := "SUM4W_VALs".Param_A413,
           OUT                      := "OUT_A413");
      A     BR;
      );
      JNB   _006;
      CALL  "HISIGMTV" (
           IN                       := "OUT_GBA25",
           STPT                     := "OUT_A413",
           PARA_VAl                 := "HISIGMTV-VALs".Param_VV2,
           OUT                      := "Z098");
_006: NOP   0;
NETWORK
TITLE = Block 273
      CALL  "HISIGMTV" (
           IN                       := "OUT_GBA26",
           STPT                     := "OUT_A413",
           PARA_VAl                 := "HISIGMTV-VALs".Param_098,
           OUT                      := "Z273");
      NOP   0;
NETWORK
TITLE = Blocks A414, 097
      A(;
      CALL  "SUM4W" (
           IN1                      := "RPCNTR",
           IN2                      := "RPTRIP5",
           IN3                      := "A50",
           IN4                      := "A50",
           PARA_VAl                 := "SUM4W_VALs".Param_A414,
           OUT                      := "OUT_A414");
      A     BR;
      );
      JNB   _007;
      CALL  "HISIGMTV" (
           IN                       := "OUT_GBA25",
           STPT                     := "OUT_A414",
           PARA_VAl                 := "HISIGMTV-VALs".Param_273,
           OUT                      := "Z097");
_007: NOP   0;
NETWORK
TITLE = Block 272
      CALL  "HISIGMTV" (
           IN                       := "OUT_GBA26",
           STPT                     := "OUT_A414",
           PARA_VAl                 := "HISIGMTV-VALs".Param_097,
           OUT                      := "ZA272");
      NOP   0;
NETWORK
TITLE = Block 003
      CALL  "QC" (
           IN                       := "OUT_GBA25",
           OUT                      := "RP1FAIL");
      NOP   0;
NETWORK
TITLE = Block 234
      CALL  "QTRANSN" (
           IN1                      := "OUT_GBA25",
           IN2                      := "OUT_GBA26",
           OUT                      := "RPOS");
      NOP   0;
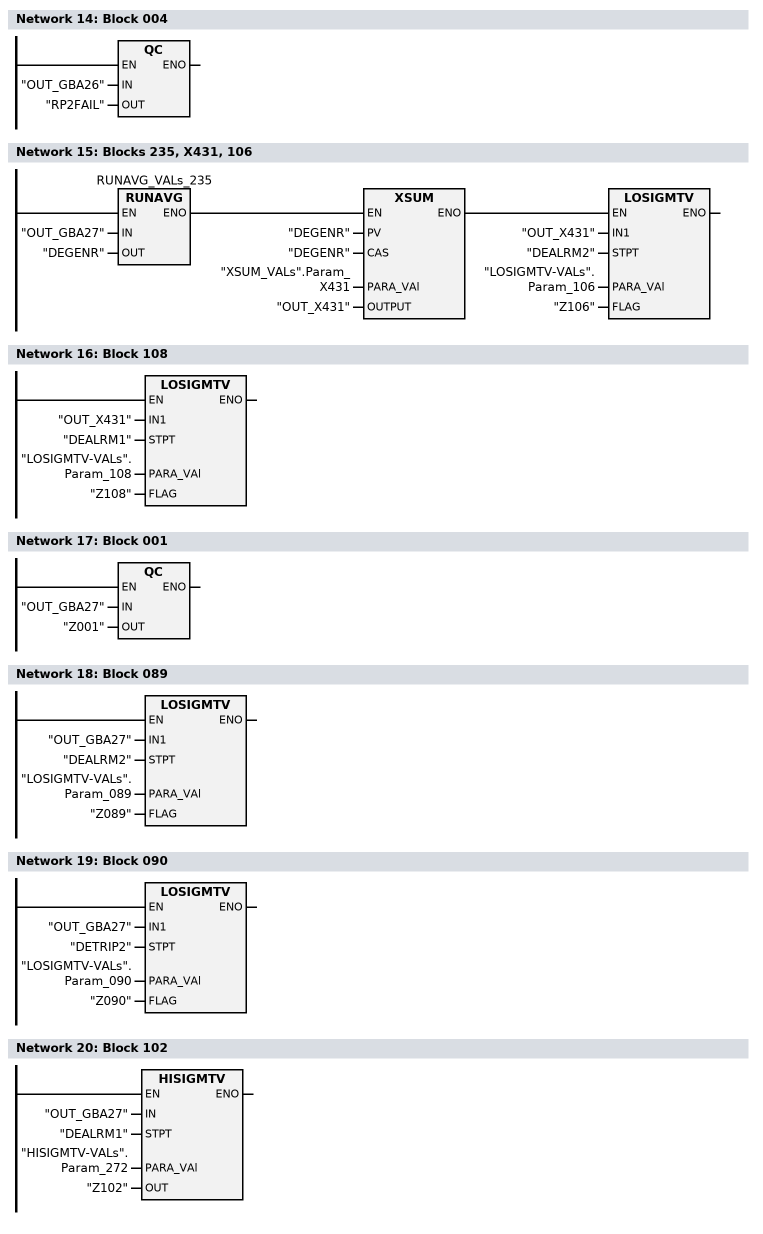
NETWORK
TITLE = Block 004
      CALL  "QC" (
           IN                       := "OUT_GBA26",
           OUT                      := "RP2FAIL");
      NOP   0;
NETWORK
TITLE = Blocks 235, X431, 106
      A(;
      A(;
      CALL  "RUNAVG" , "RUNAVG_VALs_235" (
           IN                       := "OUT_GBA27",
           OUT                      := "DEGENR");
      A     BR;
      );
      JNB   _008;
      CALL  "XSUM" (
           PV                       := "DEGENR",
           CAS                      := "DEGENR",
           PARA_VAl                 := "XSUM_VALs".Param_X431,
           OUTPUT                   := "OUT_X431");
_008: A     BR;
      );
      JNB   _009;
      CALL  "LOSIGMTV" (
           IN1                      := "OUT_X431",
           STPT                     := "DEALRM2",
           PARA_VAl                 := "LOSIGMTV-VALs".Param_106,
           FLAG                     := "Z106");
_009: NOP   0;
NETWORK
TITLE = Block 108
      CALL  "LOSIGMTV" (
           IN1                      := "OUT_X431",
           STPT                     := "DEALRM1",
           PARA_VAl                 := "LOSIGMTV-VALs".Param_108,
           FLAG                     := "Z108");
      NOP   0;
NETWORK
TITLE = Block 001
      CALL  "QC" (
           IN                       := "OUT_GBA27",
           OUT                      := "Z001");
      NOP   0;
NETWORK
TITLE = Block 089
      CALL  "LOSIGMTV" (
           IN1                      := "OUT_GBA27",
           STPT                     := "DEALRM2",
           PARA_VAl                 := "LOSIGMTV-VALs".Param_089,
           FLAG                     := "Z089");
      NOP   0;
NETWORK
TITLE = Block 090
      CALL  "LOSIGMTV" (
           IN1                      := "OUT_GBA27",
           STPT                     := "DETRIP2",
           PARA_VAl                 := "LOSIGMTV-VALs".Param_090,
           FLAG                     := "Z090");
      NOP   0;
NETWORK
TITLE = Block 102
      CALL  "HISIGMTV" (
           IN                       := "OUT_GBA27",
           STPT                     := "DEALRM1",
           PARA_VAl                 := "HISIGMTV-VALs".Param_272,
           OUT                      := "Z102");
      NOP   0;
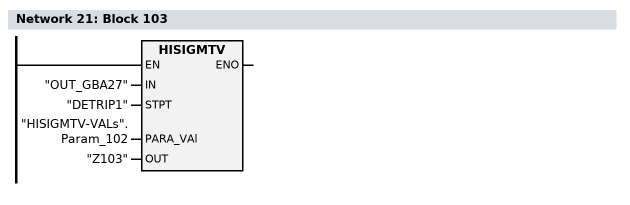
NETWORK
TITLE = Block 103
      CALL  "HISIGMTV" (
           IN                       := "OUT_GBA27",
           STPT                     := "DETRIP1",
           PARA_VAl                 := "HISIGMTV-VALs".Param_102,
           OUT                      := "Z103");
      NOP   0;
END_FUNCTION

FUNCTION "Sheet 16 (ATC)" : VOID	// FC 95
TITLE = Sheet 16 (ATC)
//ROTOR POSITION DIFFERENTIAL EXPANSION P11MXX (Digital)
AUTHOR : RJ
FAMILY : ATC
VERSION : 0.1
BEGIN
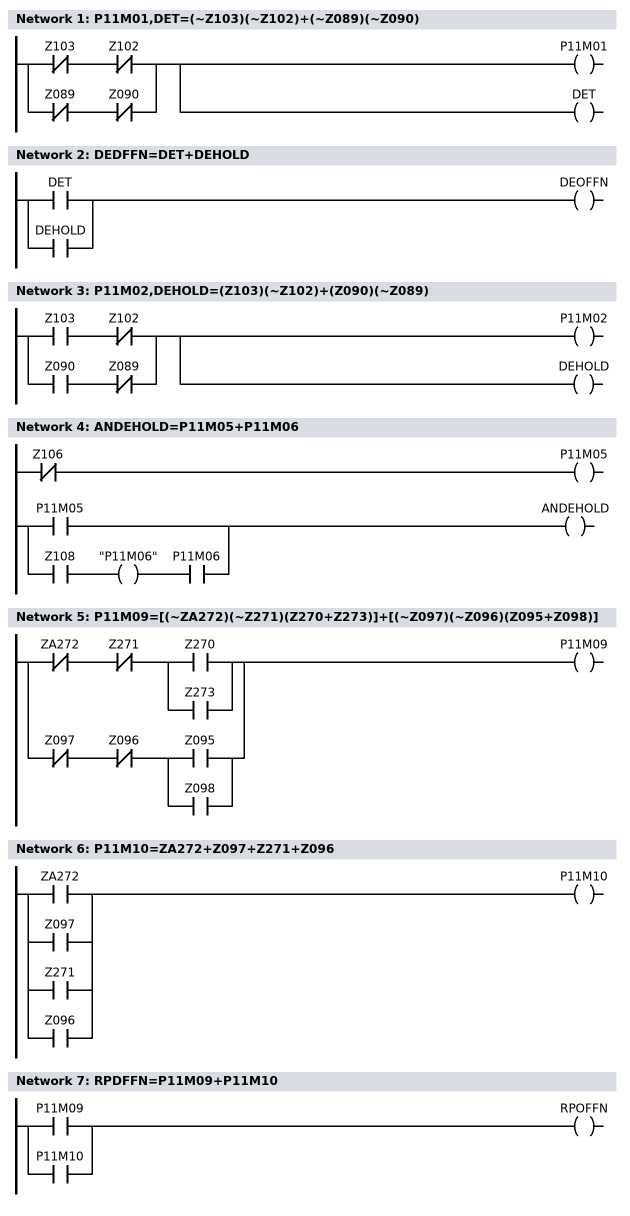
NETWORK
TITLE = P11M01,DET=(~Z103)(~Z102)+(~Z089)(~Z090)
      AN    "Z103";
      AN    "Z102";
      O;
      AN    "Z089";
      AN    "Z090";
      =     "P11M01";
      =     "DET";
NETWORK
TITLE = DEDFFN=DET+DEHOLD
      O     "DET";
      O     "DEHOLD";
      =     "DEOFFN";
NETWORK
TITLE = P11M02,DEHOLD=(Z103)(~Z102)+(Z090)(~Z089)
      A     "Z103";
      AN    "Z102";
      O;
      A     "Z090";
      AN    "Z089";
      =     "P11M02";
      =     "DEHOLD";
NETWORK
TITLE = ANDEHOLD=P11M05+P11M06
//P11M05=(~Z106)
//P11M06=Z108
      AN    "Z106";
      =     "P11M05";
      A     "P11M05";
      O(;
      A     "Z108";
      =     "P11M06";
      A     "P11M06";
      );
      =     "ANDEHOLD";
NETWORK
TITLE = P11M09=[(~ZA272)(~Z271)(Z270+Z273)]+[(~Z097)(~Z096)(Z095+Z098)]
      AN    "ZA272";
      AN    "Z271";
      A(;
      O     "Z270";
      O     "Z273";
      );
      O;
      AN    "Z097";
      AN    "Z096";
      A(;
      O     "Z095";
      O     "Z098";
      );
      =     "P11M09";
NETWORK
TITLE = P11M10=ZA272+Z097+Z271+Z096
      O     "ZA272";
      O     "Z097";
      O     "Z271";
      O     "Z096";
      =     "P11M10";
NETWORK
TITLE = RPDFFN=P11M09+P11M10
      O     "P11M09";
      O     "P11M10";
      =     "RPOFFN";
END_FUNCTION

FUNCTION "Sheet 17 (ATC)" : VOID	// FC 96
TITLE = Sheet 17 (ATC)
//LOOPS 39, 40, 41. CONDENSOR PRESS LP EXH HOOD (Analog)
AUTHOR : RJ
FAMILY : ATC
VERSION : 0.1
BEGIN
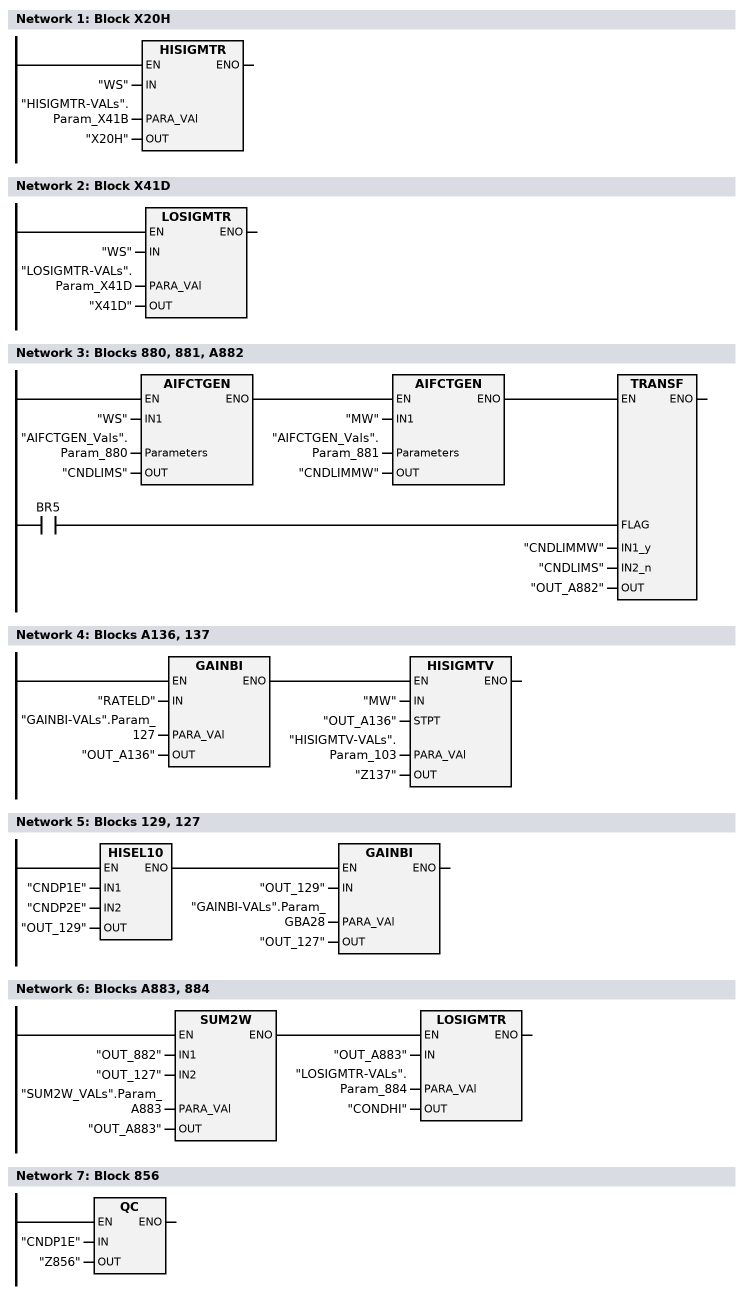
NETWORK
TITLE = Block X20H
      CALL  "HISIGMTR" (
           IN                       := "WS",
           PARA_VAl                 := "HISIGMTR-VALs".Param_X41B,
           OUT                      := "X20H");
      NOP   0;
NETWORK
TITLE = Block X41D
      CALL  "LOSIGMTR" (
           IN                       := "WS",
           PARA_VAl                 := "LOSIGMTR-VALs".Param_X41D,
           OUT                      := "X41D");
      NOP   0;
NETWORK
TITLE = Blocks 880, 881, A882
      A     "BR5";
      =     L 0.0;
      BLD   103;
      A(;
      A(;
      CALL  "AIFCTGEN" (
           IN1                      := "WS",
           Parameters               := "AIFCTGEN_Vals".Param_880,
           OUT                      := "CNDLIMS");
      A     BR;
      );
      JNB   _001;
      CALL  "AIFCTGEN" (
           IN1                      := "MW",
           Parameters               := "AIFCTGEN_Vals".Param_881,
           OUT                      := "CNDLIMMW");
_001: A     BR;
      );
      JNB   _002;
      CALL  "TRANSF" (
           FLAG                     := L 0.0,
           IN1_y                    := "CNDLIMMW",
           IN2_n                    := "CNDLIMS",
           OUT                      := "OUT_A882");
_002: NOP   0;
NETWORK
TITLE = Blocks A136, 137
      A(;
      CALL  "GAINBI" (
           IN                       := "RATELD",
           PARA_VAl                 := "GAINBI-VALs".Param_127,
           OUT                      := "OUT_A136");
      A     BR;
      );
      JNB   _003;
      CALL  "HISIGMTV" (
           IN                       := "MW",
           STPT                     := "OUT_A136",
           PARA_VAl                 := "HISIGMTV-VALs".Param_103,
           OUT                      := "Z137");
_003: NOP   0;
NETWORK
TITLE = Blocks 129, 127
      A(;
      CALL  "HISEL10" (
           IN1                      := "CNDP1E",
           IN2                      := "CNDP2E",
           OUT                      := "OUT_129");
      A     BR;
      );
      JNB   _004;
      CALL  "GAINBI" (
           IN                       := "OUT_129",
           PARA_VAl                 := "GAINBI-VALs".Param_GBA28,
           OUT                      := "OUT_127");
_004: NOP   0;
NETWORK
TITLE = Blocks A883, 884
      A(;
      CALL  "SUM2W" (
           IN1                      := "OUT_882",
           IN2                      := "OUT_127",
           PARA_VAl                 := "SUM2W_VALs".Param_A883,
           OUT                      := "OUT_A883");
      A     BR;
      );
      JNB   _005;
      CALL  "LOSIGMTR" (
           IN                       := "OUT_A883",
           PARA_VAl                 := "LOSIGMTR-VALs".Param_884,
           OUT                      := "CONDHI");
_005: NOP   0;
NETWORK
TITLE = Block 856
      CALL  "QC" (
           IN                       := "CNDP1E",
           OUT                      := "Z856");
      NOP   0;
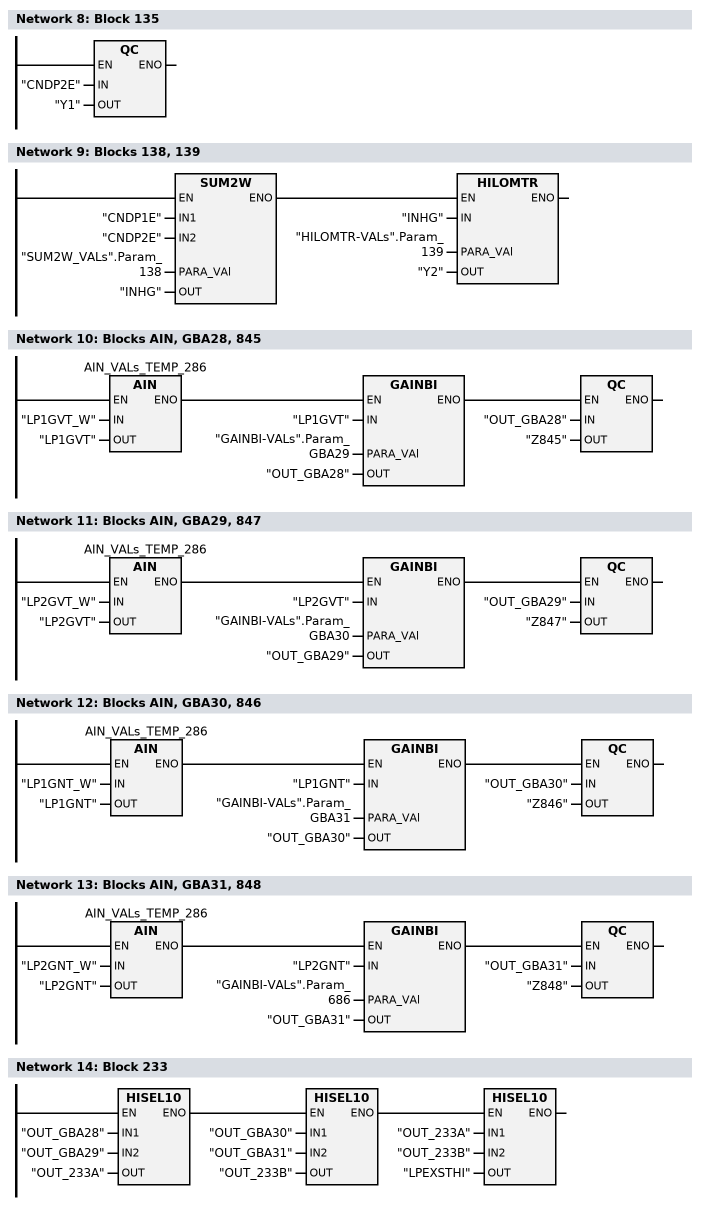
NETWORK
TITLE = Block 135
      CALL  "QC" (
           IN                       := "CNDP2E",
           OUT                      := "Y1");
      NOP   0;
NETWORK
TITLE = Blocks 138, 139
      A(;
      CALL  "SUM2W" (
           IN1                      := "CNDP1E",
           IN2                      := "CNDP2E",
           PARA_VAl                 := "SUM2W_VALs".Param_138,
           OUT                      := "INHG");
      A     BR;
      );
      JNB   _006;
      CALL  "HILOMTR" (
           IN                       := "INHG",
           PARA_VAl                 := "HILOMTR-VALs".Param_139,
           OUT                      := "Y2");
_006: NOP   0;
NETWORK
TITLE = Blocks AIN, GBA28, 845
      A(;
      A(;
      CALL  "AIN" , "AIN_VALs_TEMP_286" (
           IN                       := "LP1GVT_W",
           OUT                      := "LP1GVT");
      A     BR;
      );
      JNB   _007;
      CALL  "GAINBI" (
           IN                       := "LP1GVT",
           PARA_VAl                 := "GAINBI-VALs".Param_GBA29,
           OUT                      := "OUT_GBA28");
_007: A     BR;
      );
      JNB   _008;
      CALL  "QC" (
           IN                       := "OUT_GBA28",
           OUT                      := "Z845");
_008: NOP   0;
NETWORK
TITLE = Blocks AIN, GBA29, 847
      A(;
      A(;
      CALL  "AIN" , "AIN_VALs_TEMP_286" (
           IN                       := "LP2GVT_W",
           OUT                      := "LP2GVT");
      A     BR;
      );
      JNB   _009;
      CALL  "GAINBI" (
           IN                       := "LP2GVT",
           PARA_VAl                 := "GAINBI-VALs".Param_GBA30,
           OUT                      := "OUT_GBA29");
_009: A     BR;
      );
      JNB   _00a;
      CALL  "QC" (
           IN                       := "OUT_GBA29",
           OUT                      := "Z847");
_00a: NOP   0;
NETWORK
TITLE = Blocks AIN, GBA30, 846
      A(;
      A(;
      CALL  "AIN" , "AIN_VALs_TEMP_286" (
           IN                       := "LP1GNT_W",
           OUT                      := "LP1GNT");
      A     BR;
      );
      JNB   _00b;
      CALL  "GAINBI" (
           IN                       := "LP1GNT",
           PARA_VAl                 := "GAINBI-VALs".Param_GBA31,
           OUT                      := "OUT_GBA30");
_00b: A     BR;
      );
      JNB   _00c;
      CALL  "QC" (
           IN                       := "OUT_GBA30",
           OUT                      := "Z846");
_00c: NOP   0;
NETWORK
TITLE = Blocks AIN, GBA31, 848
      A(;
      A(;
      CALL  "AIN" , "AIN_VALs_TEMP_286" (
           IN                       := "LP2GNT_W",
           OUT                      := "LP2GNT");
      A     BR;
      );
      JNB   _00d;
      CALL  "GAINBI" (
           IN                       := "LP2GNT",
           PARA_VAl                 := "GAINBI-VALs".Param_686,
           OUT                      := "OUT_GBA31");
_00d: A     BR;
      );
      JNB   _00e;
      CALL  "QC" (
           IN                       := "OUT_GBA31",
           OUT                      := "Z848");
_00e: NOP   0;
NETWORK
TITLE = Block 233
      A(;
      A(;
      CALL  "HISEL10" (
           IN1                      := "OUT_GBA28",
           IN2                      := "OUT_GBA29",
           OUT                      := "OUT_233A");
      A     BR;
      );
      JNB   _00f;
      CALL  "HISEL10" (
           IN1                      := "OUT_GBA30",
           IN2                      := "OUT_GBA31",
           OUT                      := "OUT_233B");
_00f: A     BR;
      );
      JNB   _010;
      CALL  "HISEL10" (
           IN1                      := "OUT_233A",
           IN2                      := "OUT_233B",
           OUT                      := "LPEXSTHI");
_010: NOP   0;
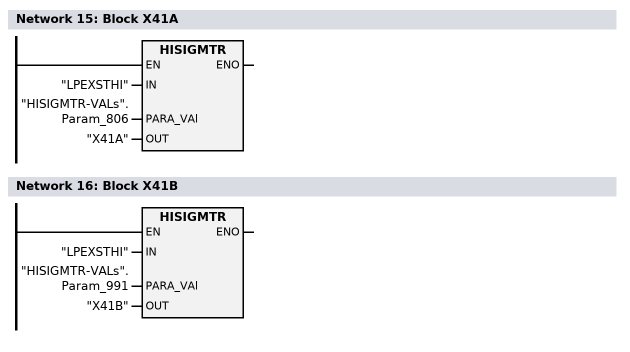
NETWORK
TITLE = Block X41A 
      CALL  "HISIGMTR" (
           IN                       := "LPEXSTHI",
           PARA_VAl                 := "HISIGMTR-VALs".Param_806,
           OUT                      := "X41A");
      NOP   0;
NETWORK
TITLE = Block X41B
      CALL  "HISIGMTR" (
           IN                       := "LPEXSTHI",
           PARA_VAl                 := "HISIGMTR-VALs".Param_991,
           OUT                      := "X41B");
      NOP   0;
END_FUNCTION

FUNCTION "Sheet 18 (ATC)" : VOID	// FC 97
TITLE = Sheet 18 (ATC)
//LADDERS 89, 90, 189, 190. GLAND, EXH, VAC - P10MXX (Digital)
AUTHOR : RJ
FAMILY : ATC
VERSION : 0.1
BEGIN
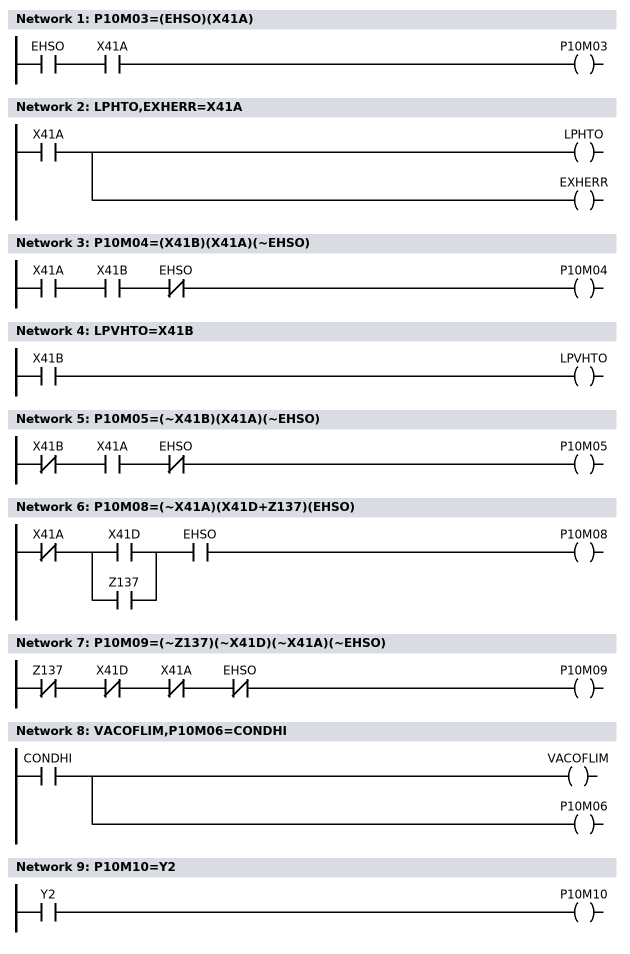
NETWORK
TITLE = P10M03=(EHSO)(X41A)
      A     "EHSO";
      A     "X41A";
      =     "P10M03";
NETWORK
TITLE = LPHTO,EXHERR=X41A
      A     "X41A";
      =     "LPHTO";
      =     "EXHERR";
NETWORK
TITLE = P10M04=(X41B)(X41A)(~EHSO)
      A     "X41A";
      A     "X41B";
      AN    "EHSO";
      =     "P10M04";
NETWORK
TITLE = LPVHTO=X41B
      A     "X41B";
      =     "LPVHTO";
NETWORK
TITLE = P10M05=(~X41B)(X41A)(~EHSO)
      AN    "X41B";
      A     "X41A";
      AN    "EHSO";
      =     "P10M05";
NETWORK
TITLE = P10M08=(~X41A)(X41D+Z137)(EHSO)
      AN    "X41A";
      A(;
      O     "X41D";
      O     "Z137";
      );
      A     "EHSO";
      =     "P10M08";
NETWORK
TITLE = P10M09=(~Z137)(~X41D)(~X41A)(~EHSO)
      AN    "Z137";
      AN    "X41D";
      AN    "X41A";
      AN    "EHSO";
      =     "P10M09";
NETWORK
TITLE = VACOFLIM,P10M06=CONDHI
      A     "CONDHI";
      =     "VACOFLIM";
      =     "P10M06";
NETWORK
TITLE = P10M10=Y2
      A     "Y2";
      =     "P10M10";
END_FUNCTION

FUNCTION "Sheet 19 (ATC)" : VOID	// FC 98
TITLE = Sheet 19 (RSM)
//BRG TEMPERATURE HIGH & VBINC (Digital)
AUTHOR : RJ
FAMILY : ATC
VERSION : 0.1
BEGIN
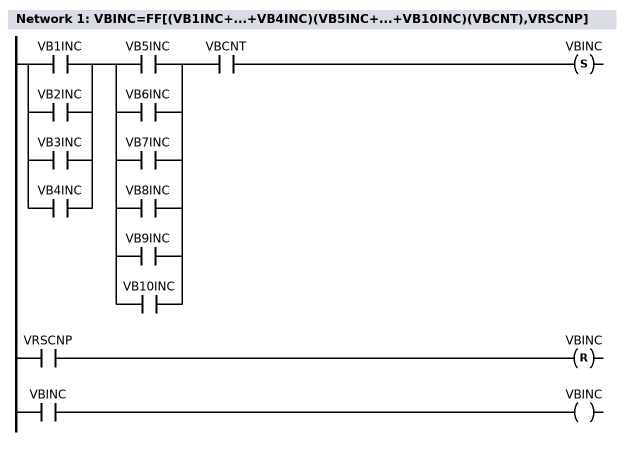
NETWORK
TITLE = VBINC=FF[(VB1INC+...+VB4INC)(VB5INC+...+VB10INC)(VBCNT),VRSCNP]
      A(;
      O     "VB1INC";
      O     "VB2INC";
      O     "VB3INC";
      O     "VB4INC";
      );
      A(;
      O     "VB5INC";
      O     "VB6INC";
      O     "VB7INC";
      O     "VB8INC";
      O     "VB9INC";
      O     "VB10INC";
      );
      A     "VBCNT";
      S     "VBINC";
      A     "VRSCNP";
      R     "VBINC";
      A     "VBINC";
      =     "VBINC";
END_FUNCTION

FUNCTION "Sheet 20 (ATC)" : VOID	// FC 99
TITLE = Sheet 20 (ATC)
//VIBRATION LIMIT (Analog)
AUTHOR : RJ
FAMILY : ATC
VERSION : 0.1
BEGIN
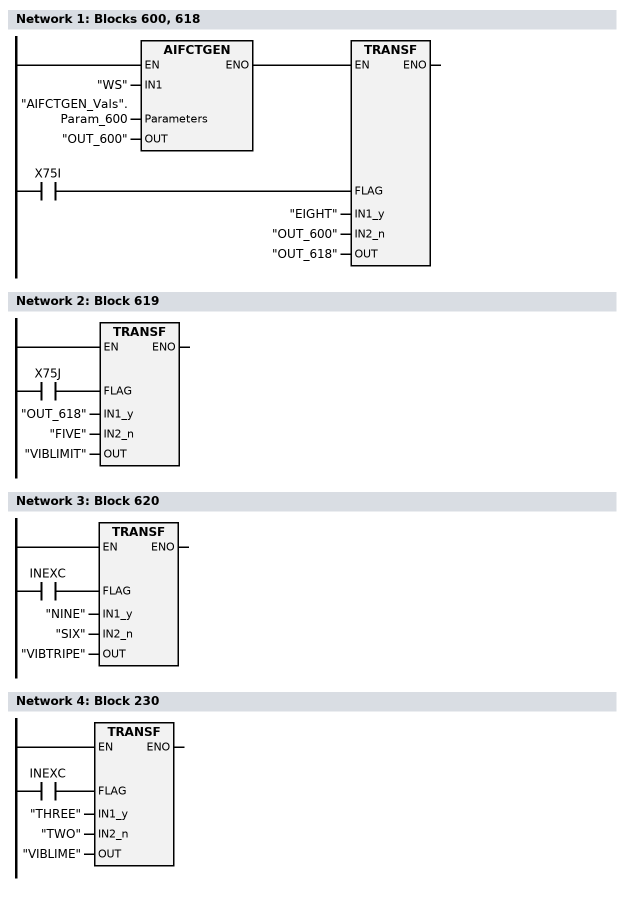
NETWORK
TITLE = Blocks 600, 618
      A     "X75I";
      =     L 0.0;
      BLD   103;
      A(;
      CALL  "AIFCTGEN" (
           IN1                      := "WS",
           Parameters               := "AIFCTGEN_Vals".Param_600,
           OUT                      := "OUT_600");
      A     BR;
      );
      JNB   _001;
      CALL  "TRANSF" (
           FLAG                     := L 0.0,
           IN1_y                    := "EIGHT",
           IN2_n                    := "OUT_600",
           OUT                      := "OUT_618");
_001: NOP   0;
NETWORK
TITLE = Block 619
      A     "X75J";
      =     L 0.0;
      BLD   103;
      CALL  "TRANSF" (
           FLAG                     := L 0.0,
           IN1_y                    := "OUT_618",
           IN2_n                    := "FIVE",
           OUT                      := "VIBLIMIT");
      NOP   0;
NETWORK
TITLE = Block 620
      A     "INEXC";
      =     L 0.0;
      BLD   103;
      CALL  "TRANSF" (
           FLAG                     := L 0.0,
           IN1_y                    := "NINE",
           IN2_n                    := "SIX",
           OUT                      := "VIBTRIPE");
      NOP   0;
NETWORK
TITLE = Block 230
      A     "INEXC";
      =     L 0.0;
      BLD   103;
      CALL  "TRANSF" (
           FLAG                     := L 0.0,
           IN1_y                    := "THREE",
           IN2_n                    := "TWO",
           OUT                      := "VIBLIME");
      NOP   0;
END_FUNCTION

FUNCTION "Sheet 21 (ATC)" : VOID	// FC 100
TITLE = Sheet 21 (ATC)
//LADDERS 302,304,306,400. VIBRATION ALARM AND TRIP (Digital)
AUTHOR : RJ
FAMILY : ATC
VERSION : 0.1
BEGIN
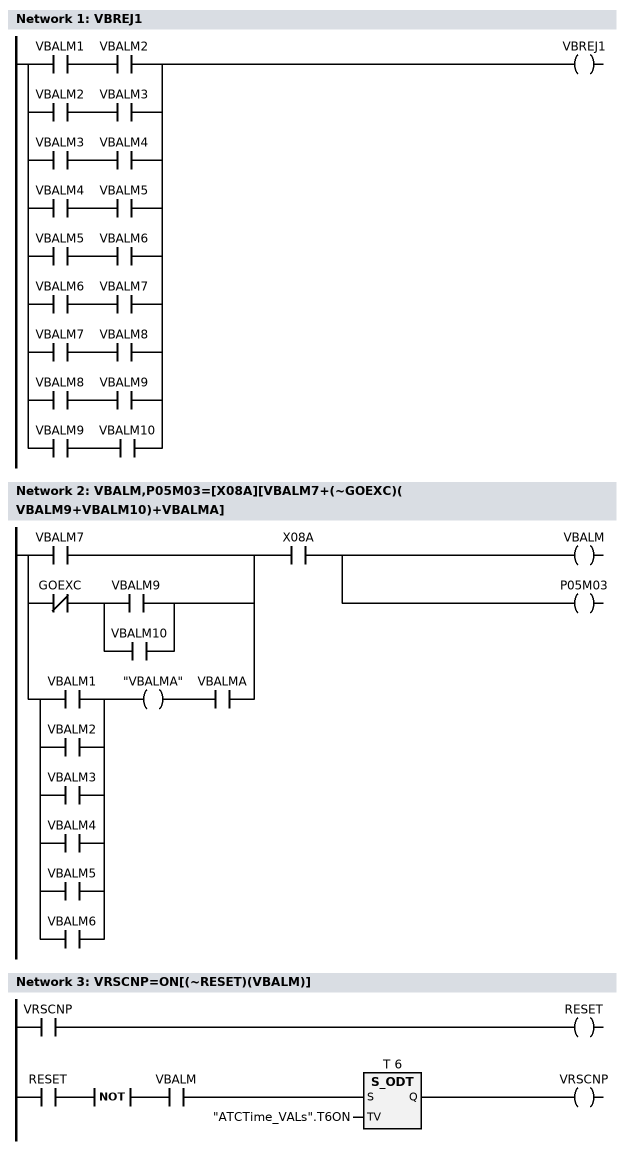
NETWORK
TITLE = VBREJ1
//VBREJ1=[(VBALM1)(VBALM2)]+[(VBALM2)(VBALM3)]+...+[(VBALM9)(VBALM10)]
//
      A     "VBALM1";
      A     "VBALM2";
      O;
      A     "VBALM2";
      A     "VBALM3";
      O;
      A     "VBALM3";
      A     "VBALM4";
      O;
      A     "VBALM4";
      A     "VBALM5";
      O;
      A     "VBALM5";
      A     "VBALM6";
      O;
      A     "VBALM6";
      A     "VBALM7";
      O;
      A     "VBALM7";
      A     "VBALM8";
      O;
      A     "VBALM8";
      A     "VBALM9";
      O;
      A     "VBALM9";
      A     "VBALM10";
      =     "VBREJ1";
NETWORK
TITLE = VBALM,P05M03=[X08A][VBALM7+(~GOEXC)(VBALM9+VBALM10)+VBALMA]
//VBALMA=VBALM1+VBALM2+...+VBALM6
      A(;
      O     "VBALM7";
      O(;
      AN    "GOEXC";
      A(;
      O     "VBALM9";
      O     "VBALM10";
      );
      );
      O(;
      A(;
      O     "VBALM1";
      O     "VBALM2";
      O     "VBALM3";
      O     "VBALM4";
      O     "VBALM5";
      O     "VBALM6";
      );
      =     "VBALMA";
      A     "VBALMA";
      );
      );
      A     "X08A";
      =     "VBALM";
      =     "P05M03";
NETWORK
TITLE = VRSCNP=ON[(~RESET)(VBALM)]
//RESET=VRSCNP
      A     "VRSCNP";
      =     "RESET";
      A     "RESET";
      NOT;
      A     "VBALM";
      L     "ATCTime_VALs".T6ON;
      SD    T 6;
      NOP   0;
      NOP   0;
      NOP   0;
      A     T 6;
      =     "VRSCNP";
